// Mitsubishi GX Developer project: 11-1105_20130914   PLC: FX3U

PROGRAM MAIN
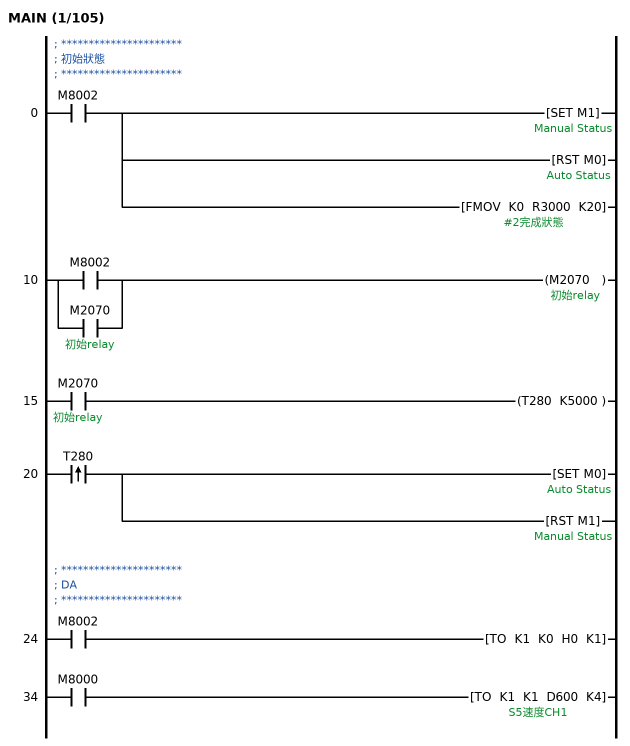
; **********************
; 初始狀態
; **********************
0     LD      M8002
      SET     M1  ; Manual Status
      RST     M0  ; Auto Status
      FMOV    K0 R3000 K20  ; #2完成狀態
10    LD      M8002
      OR      M2070  ; 初始relay
      OUT     M2070  ; 初始relay
15    LD      M2070  ; 初始relay
      OUT     T280 K5000
20    LDP     T280
      SET     M0  ; Auto Status
      RST     M1  ; Manual Status
; **********************
; DA
; **********************
24    LD      M8002
      TO      K1 K0 H0 K1
34    LD      M8000
      TO      K1 K1 D600 K4  ; S5速度CH1
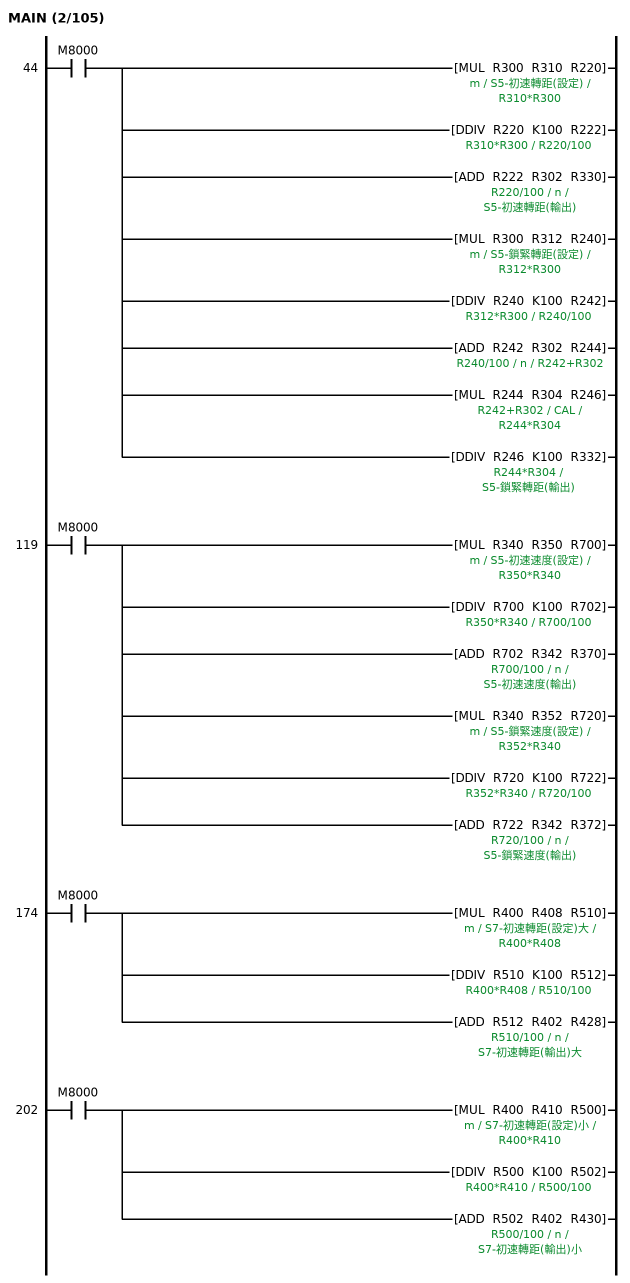
44    LD      M8000
      MUL     R300 R310 R220  ; m / S5-初速轉距(設定) / R310*R300
      DDIV    R220 K100 R222  ; R220/100
      ADD     R222 R302 R330  ; n / S5-初速轉距(輸出)
      MUL     R300 R312 R240  ; S5-鎖緊轉距(設定) / R312*R300
      DDIV    R240 K100 R242  ; R240/100
      ADD     R242 R302 R244  ; R242+R302
      MUL     R244 R304 R246  ; CAL / R244*R304
      DDIV    R246 K100 R332  ; S5-鎖緊轉距(輸出)
119   LD      M8000
      MUL     R340 R350 R700  ; m / S5-初速速度(設定) / R350*R340
      DDIV    R700 K100 R702  ; R700/100
      ADD     R702 R342 R370  ; n / S5-初速速度(輸出)
      MUL     R340 R352 R720  ; S5-鎖緊速度(設定) / R352*R340
      DDIV    R720 K100 R722  ; R720/100
      ADD     R722 R342 R372  ; S5-鎖緊速度(輸出)
174   LD      M8000
      MUL     R400 R408 R510  ; m / S7-初速轉距(設定)大 / R400*R408
      DDIV    R510 K100 R512  ; R510/100
      ADD     R512 R402 R428  ; n / S7-初速轉距(輸出)大
202   LD      M8000
      MUL     R400 R410 R500  ; S7-初速轉距(設定)小 / R400*R410
      DDIV    R500 K100 R502  ; R500/100
      ADD     R502 R402 R430  ; S7-初速轉距(輸出)小
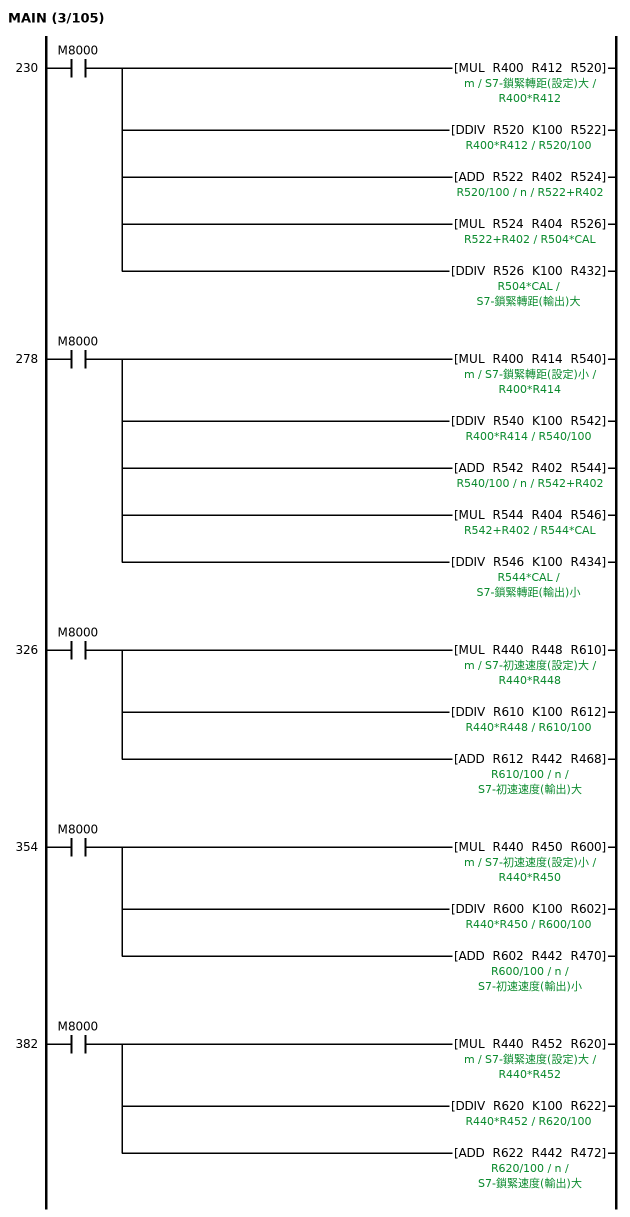
230   LD      M8000
      MUL     R400 R412 R520  ; S7-鎖緊轉距(設定)大 / R400*R412
      DDIV    R520 K100 R522  ; R520/100
      ADD     R522 R402 R524  ; R522+R402
      MUL     R524 R404 R526  ; R504*CAL
      DDIV    R526 K100 R432  ; S7-鎖緊轉距(輸出)大
278   LD      M8000
      MUL     R400 R414 R540  ; S7-鎖緊轉距(設定)小 / R400*R414
      DDIV    R540 K100 R542  ; R540/100
      ADD     R542 R402 R544  ; R542+R402
      MUL     R544 R404 R546  ; R544*CAL
      DDIV    R546 K100 R434  ; S7-鎖緊轉距(輸出)小
326   LD      M8000
      MUL     R440 R448 R610  ; m / S7-初速速度(設定)大 / R440*R448
      DDIV    R610 K100 R612  ; R610/100
      ADD     R612 R442 R468  ; n / S7-初速速度(輸出)大
354   LD      M8000
      MUL     R440 R450 R600  ; S7-初速速度(設定)小 / R440*R450
      DDIV    R600 K100 R602  ; R600/100
      ADD     R602 R442 R470  ; S7-初速速度(輸出)小
382   LD      M8000
      MUL     R440 R452 R620  ; S7-鎖緊速度(設定)大 / R440*R452
      DDIV    R620 K100 R622  ; R620/100
      ADD     R622 R442 R472  ; S7-鎖緊速度(輸出)大
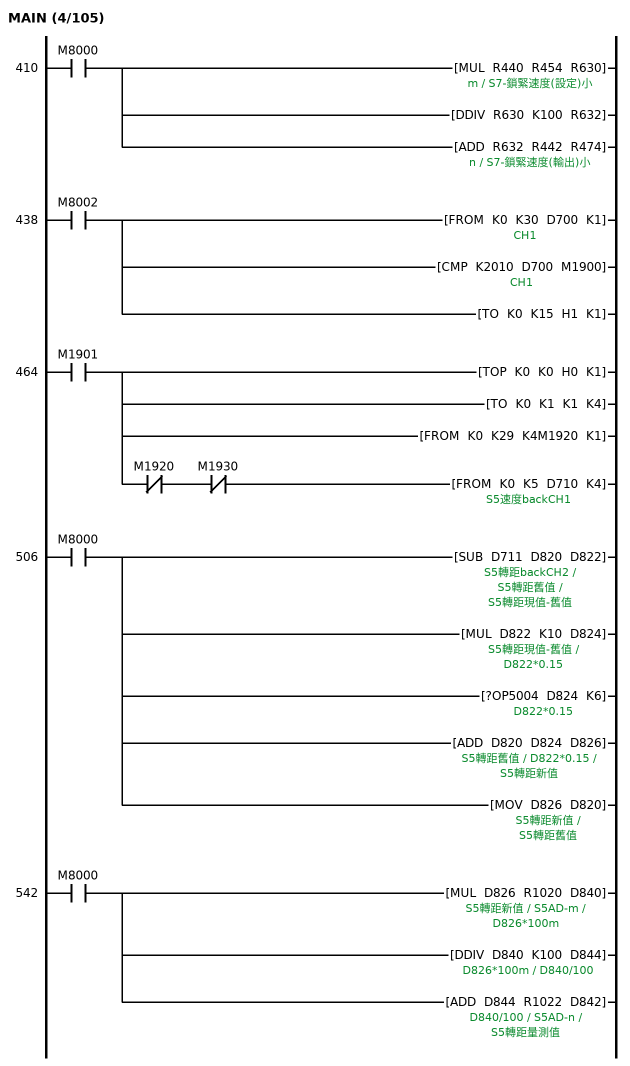
410   LD      M8000
      MUL     R440 R454 R630  ; S7-鎖緊速度(設定)小
      DDIV    R630 K100 R632
      ADD     R632 R442 R474  ; S7-鎖緊速度(輸出)小
438   LD      M8002
      FROM    K0 K30 D700 K1  ; CH1
      CMP     K2010 D700 M1900
      TO      K0 K15 H1 K1
464   LD      M1901
      TOP     K0 K0 H0 K1
      TO      K0 K1 K1 K4
      FROM    K0 K29 K4M1920 K1
      ANI     M1920
      ANI     M1930
      FROM    K0 K5 D710 K4  ; S5速度backCH1
506   LD      M8000
      SUB     D711 D820 D822  ; S5轉距backCH2 / S5轉距舊值 / S5轉距現值-舊值
      MUL     D822 K10 D824  ; D822*0.15
      ?OP5004 D824 K6
      ADD     D820 D824 D826  ; S5轉距新值
      MOV     D826 D820
542   LD      M8000
      MUL     D826 R1020 D840  ; S5AD-m / D826*100m
      DDIV    D840 K100 D844  ; D840/100
      ADD     D844 R1022 D842  ; S5AD-n / S5轉距量測值
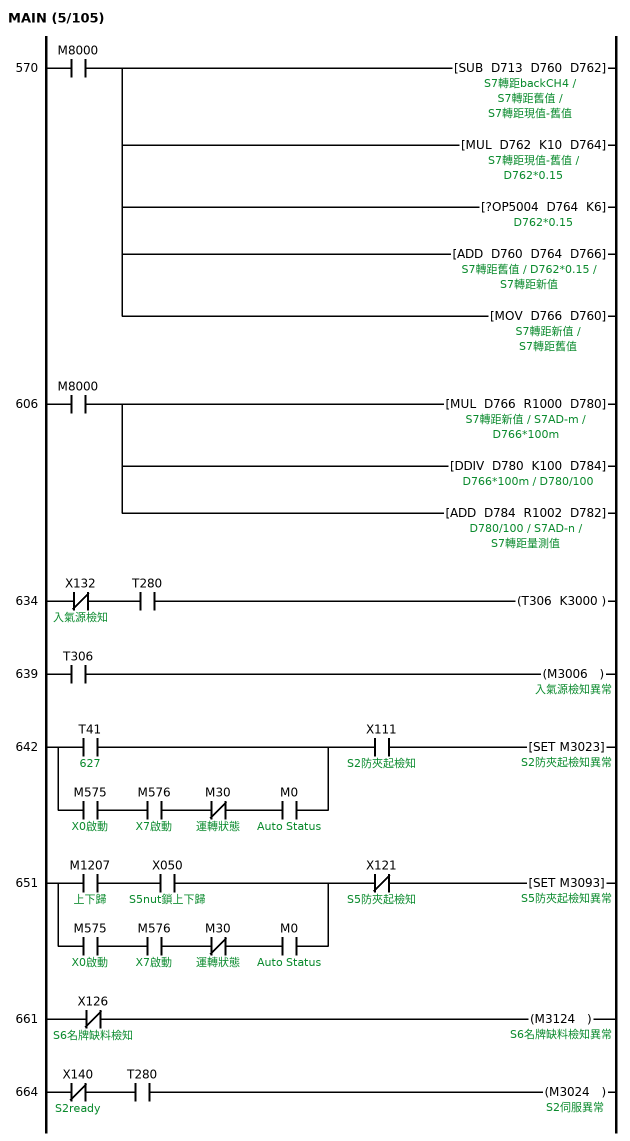
570   LD      M8000
      SUB     D713 D760 D762  ; S7轉距backCH4 / S7轉距舊值 / S7轉距現值-舊值
      MUL     D762 K10 D764  ; D762*0.15
      ?OP5004 D764 K6
      ADD     D760 D764 D766  ; S7轉距新值
      MOV     D766 D760
606   LD      M8000
      MUL     D766 R1000 D780  ; S7AD-m / D766*100m
      DDIV    D780 K100 D784  ; D780/100
      ADD     D784 R1002 D782  ; S7AD-n / S7轉距量測值
634   LDI     X132  ; 入氣源檢知
      AND     T280
      OUT     T306 K3000
639   LD      T306
      OUT     M3006  ; 入氣源檢知異常
642   LD      T41  ; 627
      LD      M575  ; X0啟動
      AND     M576  ; X7啟動
      ANI     M30  ; 運轉狀態
      AND     M0  ; Auto Status
      ORB
      AND     X111  ; S2防夾起檢知
      SET     M3023  ; S2防夾起檢知異常
651   LD      M1207  ; 上下歸
      AND     X050  ; S5nut鎖上下歸
      LD      M575  ; X0啟動
      AND     M576  ; X7啟動
      ANI     M30  ; 運轉狀態
      AND     M0  ; Auto Status
      ORB
      ANI     X121  ; S5防夾起檢知
      SET     M3093  ; S5防夾起檢知異常
661   LDI     X126  ; S6名牌缺料檢知
      OUT     M3124  ; S6名牌缺料檢知異常
664   LDI     X140  ; S2ready
      AND     T280
      OUT     M3024  ; S2伺服異常
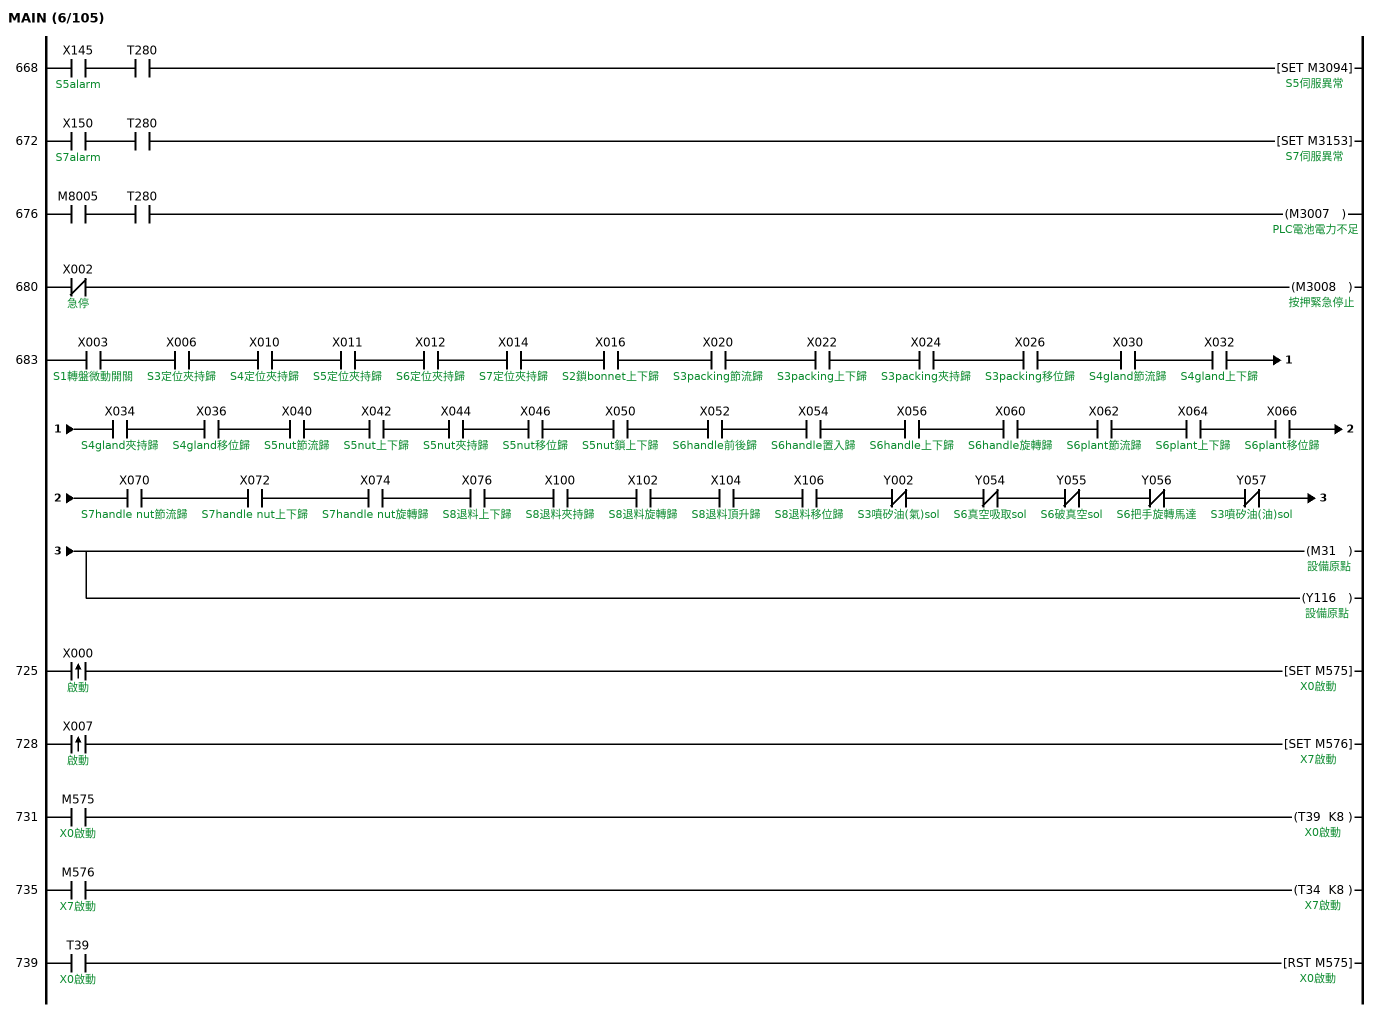
668   LD      X145  ; S5alarm
      AND     T280
      SET     M3094  ; S5伺服異常
672   LD      X150  ; S7alarm
      AND     T280
      SET     M3153  ; S7伺服異常
676   LD      M8005
      AND     T280
      OUT     M3007  ; PLC電池電力不足
680   LDI     X002  ; 急停
      OUT     M3008  ; 按押緊急停止
683   LD      X003  ; S1轉盤微動開關
      AND     X006  ; S3定位夾持歸
      AND     X010  ; S4定位夾持歸
      AND     X011  ; S5定位夾持歸
      AND     X012  ; S6定位夾持歸
      AND     X014  ; S7定位夾持歸
      AND     X016  ; S2鎖bonnet上下歸
      AND     X020  ; S3packing節流歸
      AND     X022  ; S3packing上下歸
      AND     X024  ; S3packing夾持歸
      AND     X026  ; S3packing移位歸
      AND     X030  ; S4gland節流歸
      AND     X032  ; S4gland上下歸
      AND     X034  ; S4gland夾持歸
      AND     X036  ; S4gland移位歸
      AND     X040  ; S5nut節流歸
      AND     X042  ; S5nut上下歸
      AND     X044  ; S5nut夾持歸
      AND     X046  ; S5nut移位歸
      AND     X050  ; S5nut鎖上下歸
      AND     X052  ; S6handle前後歸
      AND     X054  ; S6handle置入歸
      AND     X056  ; S6handle上下歸
      AND     X060  ; S6handle旋轉歸
      AND     X062  ; S6plant節流歸
      AND     X064  ; S6plant上下歸
      AND     X066  ; S6plant移位歸
      AND     X070  ; S7handle nut節流歸
      AND     X072  ; S7handle nut上下歸
      AND     X074  ; S7handle nut旋轉歸
      AND     X076  ; S8退料上下歸
      AND     X100  ; S8退料夾持歸
      AND     X102  ; S8退料旋轉歸
      AND     X104  ; S8退料頂升歸
      AND     X106  ; S8退料移位歸
      ANI     Y002  ; S3噴矽油(氣)sol
      ANI     Y054  ; S6真空吸取sol
      ANI     Y055  ; S6破真空sol
      ANI     Y056  ; S6把手旋轉馬達
      ANI     Y057  ; S3噴矽油(油)sol
      OUT     M31  ; 設備原點
      OUT     Y116  ; 設備原點
725   LDP     X000  ; 啟動
      SET     M575  ; X0啟動
728   LDP     X007  ; 啟動
      SET     M576  ; X7啟動
731   LD      M575  ; X0啟動
      OUT     T39 K8  ; X0啟動
735   LD      M576  ; X7啟動
      OUT     T34 K8  ; X7啟動
739   LD      T39  ; X0啟動
      RST     M575  ; X0啟動
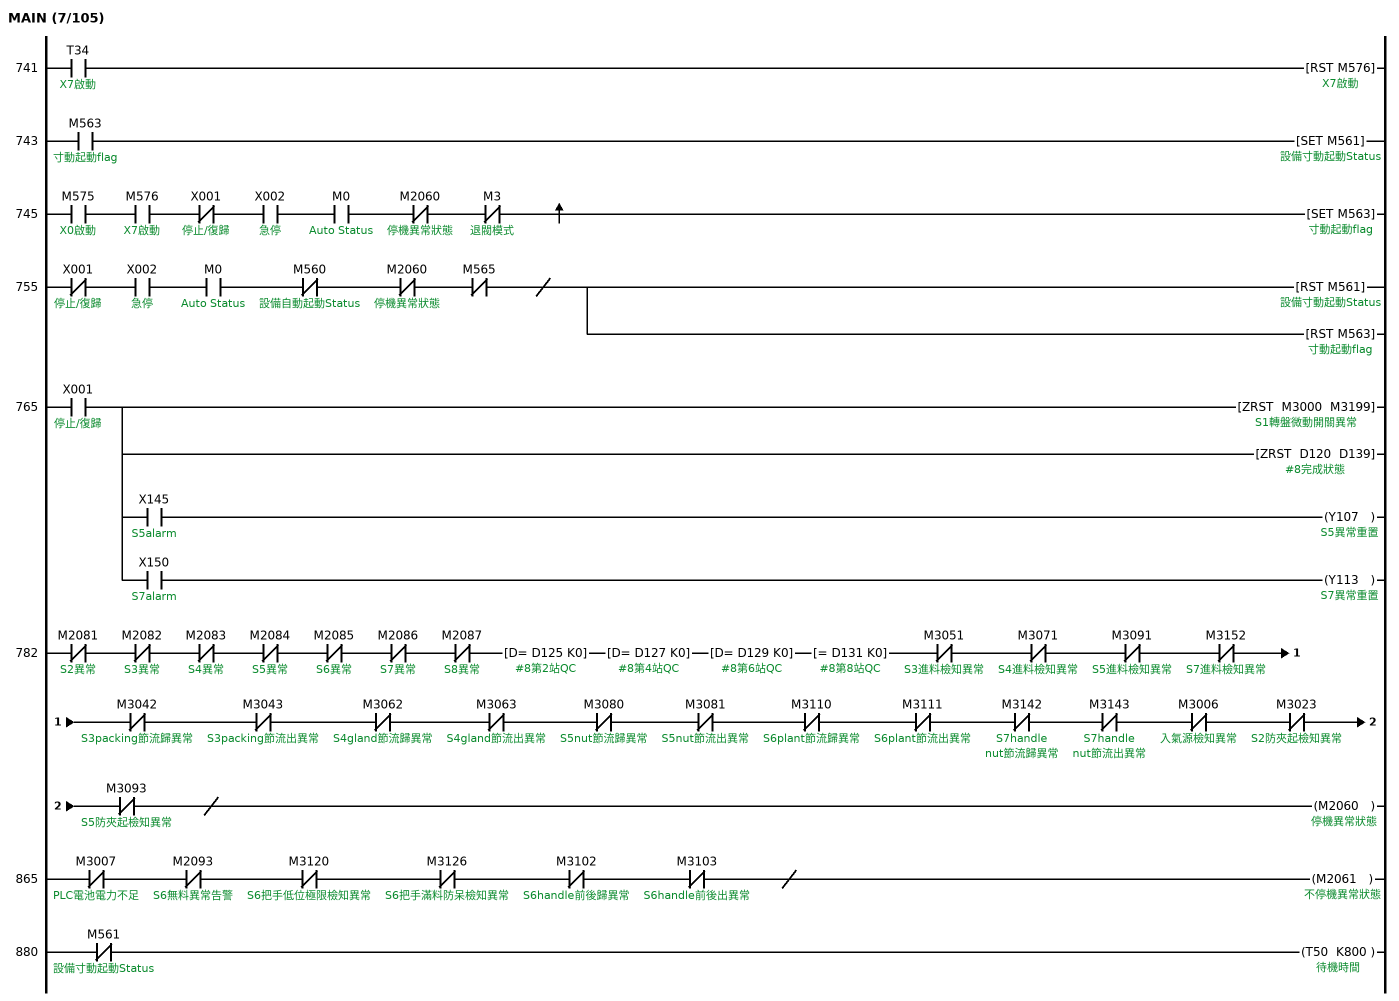
741   LD      T34  ; X7啟動
      RST     M576  ; X7啟動
743   LD      M563  ; 寸動起動flag
      SET     M561  ; 設備寸動起動Status
745   LD      M575  ; X0啟動
      AND     M576  ; X7啟動
      ANI     X001  ; 停止/復歸
      AND     X002  ; 急停
      AND     M0  ; Auto Status
      ANI     M2060  ; 停機異常狀態
      ANI     M3  ; 退閥模式
      MEP
      SET     M563  ; 寸動起動flag
755   LDI     X001  ; 停止/復歸
      AND     X002  ; 急停
      AND     M0  ; Auto Status
      ANI     M560  ; 設備自動起動Status
      ANI     M2060  ; 停機異常狀態
      ANI     M565
      INV
      RST     M561  ; 設備寸動起動Status
      RST     M563  ; 寸動起動flag
765   LD      X001  ; 停止/復歸
      ZRST    M3000 M3199  ; S1轉盤微動開關異常
      ZRST    D120 D139  ; #8完成狀態
      MPS
      AND     X145  ; S5alarm
      OUT     Y107  ; S5異常重置
      MPP
      AND     X150  ; S7alarm
      OUT     Y113  ; S7異常重置
782   LDI     M2081  ; S2異常
      ANI     M2082  ; S3異常
      ANI     M2083  ; S4異常
      ANI     M2084  ; S5異常
      ANI     M2085  ; S6異常
      ANI     M2086  ; S7異常
      ANI     M2087  ; S8異常
      ANDD=   D125 K0  ; #8第2站QC
      ANDD=   D127 K0  ; #8第4站QC
      ANDD=   D129 K0  ; #8第6站QC
      AND=    D131 K0  ; #8第8站QC
      ANI     M3051  ; S3進料檢知異常
      ANI     M3071  ; S4進料檢知異常
      ANI     M3091  ; S5進料檢知異常
      ANI     M3152  ; S7進料檢知異常
      ANI     M3042  ; S3packing節流歸異常
      ANI     M3043  ; S3packing節流出異常
      ANI     M3062  ; S4gland節流歸異常
      ANI     M3063  ; S4gland節流出異常
      ANI     M3080  ; S5nut節流歸異常
      ANI     M3081  ; S5nut節流出異常
      ANI     M3110  ; S6plant節流歸異常
      ANI     M3111  ; S6plant節流出異常
      ANI     M3142  ; S7handle nut節流歸異常
      ANI     M3143  ; S7handle nut節流出異常
      ANI     M3006  ; 入氣源檢知異常
      ANI     M3023  ; S2防夾起檢知異常
      ANI     M3093  ; S5防夾起檢知異常
      INV
      OUT     M2060  ; 停機異常狀態
865   LDI     M3007  ; PLC電池電力不足
      ANI     M2093  ; S6無料異常告警
      ANI     M3120  ; S6把手低位極限檢知異常
      ANI     M3126  ; S6把手滿料防呆檢知異常
      ANI     M3102  ; S6handle前後歸異常
      ANI     M3103  ; S6handle前後出異常
      INV
      OUT     M2061  ; 不停機異常狀態
880   LDI     M561  ; 設備寸動起動Status
      OUT     T50 K800  ; 待機時間
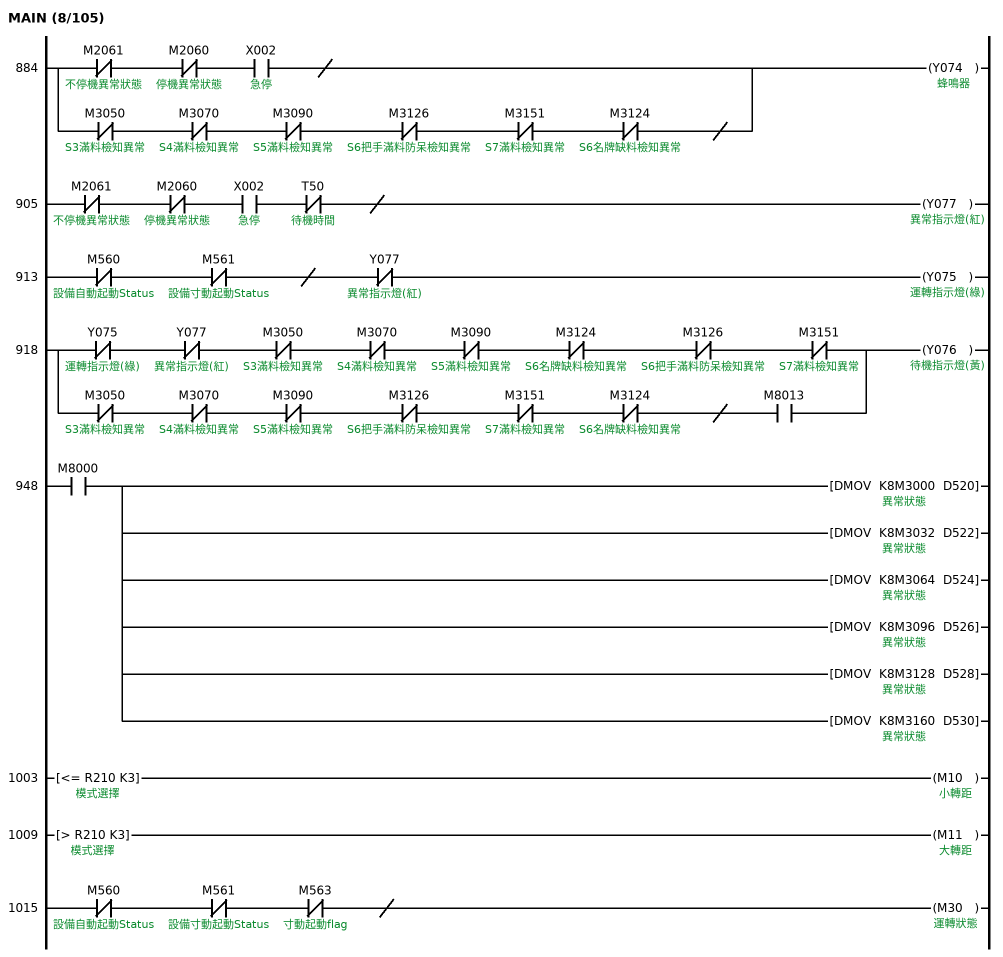
884   LDI     M2061  ; 不停機異常狀態
      ANI     M2060  ; 停機異常狀態
      AND     X002  ; 急停
      INV
      LDI     M3050  ; S3滿料檢知異常
      ANI     M3070  ; S4滿料檢知異常
      ANI     M3090  ; S5滿料檢知異常
      ANI     M3126  ; S6把手滿料防呆檢知異常
      ANI     M3151  ; S7滿料檢知異常
      ANI     M3124  ; S6名牌缺料檢知異常
      INV
      ORB
      OUT     Y074  ; 蜂鳴器
905   LDI     M2061  ; 不停機異常狀態
      ANI     M2060  ; 停機異常狀態
      AND     X002  ; 急停
      ANI     T50  ; 待機時間
      INV
      OUT     Y077  ; 異常指示燈(紅)
913   LDI     M560  ; 設備自動起動Status
      ANI     M561  ; 設備寸動起動Status
      INV
      ANI     Y077  ; 異常指示燈(紅)
      OUT     Y075  ; 運轉指示燈(綠)
918   LDI     Y075  ; 運轉指示燈(綠)
      ANI     Y077  ; 異常指示燈(紅)
      ANI     M3050  ; S3滿料檢知異常
      ANI     M3070  ; S4滿料檢知異常
      ANI     M3090  ; S5滿料檢知異常
      ANI     M3124  ; S6名牌缺料檢知異常
      ANI     M3126  ; S6把手滿料防呆檢知異常
      ANI     M3151  ; S7滿料檢知異常
      LDI     M3050  ; S3滿料檢知異常
      ANI     M3070  ; S4滿料檢知異常
      ANI     M3090  ; S5滿料檢知異常
      ANI     M3126  ; S6把手滿料防呆檢知異常
      ANI     M3151  ; S7滿料檢知異常
      ANI     M3124  ; S6名牌缺料檢知異常
      INV
      AND     M8013
      ORB
      OUT     Y076  ; 待機指示燈(黃)
948   LD      M8000
      DMOV    K8M3000 D520  ; 異常狀態
      DMOV    K8M3032 D522  ; 異常狀態
      DMOV    K8M3064 D524  ; S4gland上下歸異常 / 異常狀態
      DMOV    K8M3096 D526  ; S4定位夾持歸異常 / 異常狀態
      DMOV    K8M3128 D528  ; 異常狀態
      DMOV    K8M3160 D530  ; S8退料上下歸異常 / 異常狀態
1003  LD<=    R210 K3  ; 模式選擇
      OUT     M10  ; 小轉距
1009  LD>     R210 K3  ; 模式選擇
      OUT     M11  ; 大轉距
1015  LDI     M560  ; 設備自動起動Status
      ANI     M561  ; 設備寸動起動Status
      ANI     M563  ; 寸動起動flag
      INV
      OUT     M30  ; 運轉狀態
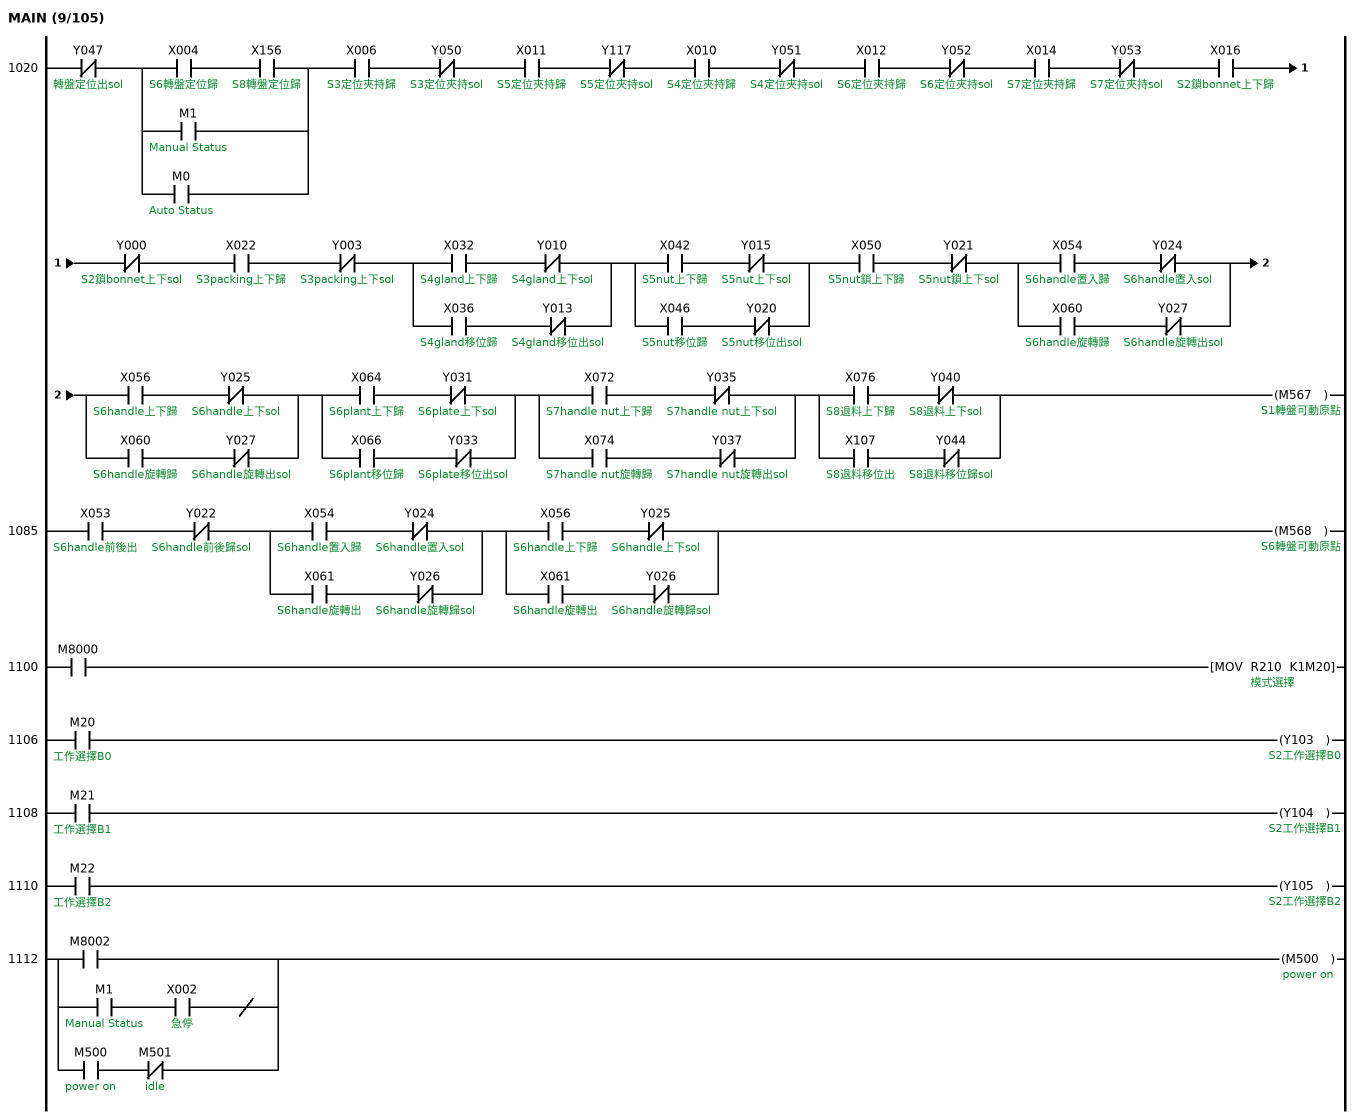
1020  LDI     Y047  ; 轉盤定位出sol
      LD      X004  ; S6轉盤定位歸
      AND     X156  ; S8轉盤定位歸
      OR      M1  ; Manual Status
      OR      M0  ; Auto Status
      ANB
      AND     X006  ; S3定位夾持歸
      ANI     Y050  ; S3定位夾持sol
      AND     X011  ; S5定位夾持歸
      ANI     Y117  ; S5定位夾持sol
      AND     X010  ; S4定位夾持歸
      ANI     Y051  ; S4定位夾持sol
      AND     X012  ; S6定位夾持歸
      ANI     Y052  ; S6定位夾持sol
      AND     X014  ; S7定位夾持歸
      ANI     Y053  ; S7定位夾持sol
      AND     X016  ; S2鎖bonnet上下歸
      ANI     Y000  ; S2鎖bonnet上下sol
      AND     X022  ; S3packing上下歸
      ANI     Y003  ; S3packing上下sol
      LD      X032  ; S4gland上下歸
      ANI     Y010  ; S4gland上下sol
      LD      X036  ; S4gland移位歸
      ANI     Y013  ; S4gland移位出sol
      ORB
      ANB
      LD      X042  ; S5nut上下歸
      ANI     Y015  ; S5nut上下sol
      LD      X046  ; S5nut移位歸
      ANI     Y020  ; S5nut移位出sol
      ORB
      ANB
      AND     X050  ; S5nut鎖上下歸
      ANI     Y021  ; S5nut鎖上下sol
      LD      X054  ; S6handle置入歸
      ANI     Y024  ; S6handle置入sol
      LD      X060  ; S6handle旋轉歸
      ANI     Y027  ; S6handle旋轉出sol
      ORB
      ANB
      LD      X056  ; S6handle上下歸
      ANI     Y025  ; S6handle上下sol
      LD      X060  ; S6handle旋轉歸
      ANI     Y027  ; S6handle旋轉出sol
      ORB
      ANB
      LD      X064  ; S6plant上下歸
      ANI     Y031  ; S6plate上下sol
      LD      X066  ; S6plant移位歸
      ANI     Y033  ; S6plate移位出sol
      ORB
      ANB
      LD      X072  ; S7handle nut上下歸
      ANI     Y035  ; S7handle nut上下sol
      LD      X074  ; S7handle nut旋轉歸
      ANI     Y037  ; S7handle nut旋轉出sol
      ORB
      ANB
      LD      X076  ; S8退料上下歸
      ANI     Y040  ; S8退料上下sol
      LD      X107  ; S8退料移位出
      ANI     Y044  ; S8退料移位歸sol
      ORB
      ANB
      OUT     M567  ; S1轉盤可動原點
1085  LD      X053  ; S6handle前後出
      ANI     Y022  ; S6handle前後歸sol
      LD      X054  ; S6handle置入歸
      ANI     Y024  ; S6handle置入sol
      LD      X061  ; S6handle旋轉出
      ANI     Y026  ; S6handle旋轉歸sol
      ORB
      ANB
      LD      X056  ; S6handle上下歸
      ANI     Y025  ; S6handle上下sol
      LD      X061  ; S6handle旋轉出
      ANI     Y026  ; S6handle旋轉歸sol
      ORB
      ANB
      OUT     M568  ; S6轉盤可動原點
1100  LD      M8000
      MOV     R210 K1M20  ; 工作選擇B0
1106  LD      M20  ; 工作選擇B0
      OUT     Y103  ; S2工作選擇B0
1108  LD      M21  ; 工作選擇B1
      OUT     Y104  ; S2工作選擇B1
1110  LD      M22  ; 工作選擇B2
      OUT     Y105  ; S2工作選擇B2
1112  LD      M8002
      LD      M1  ; Manual Status
      AND     X002  ; 急停
      INV
      ORB
      LD      M500  ; power on
      ANI     M501  ; idle
      ORB
      OUT     M500  ; power on
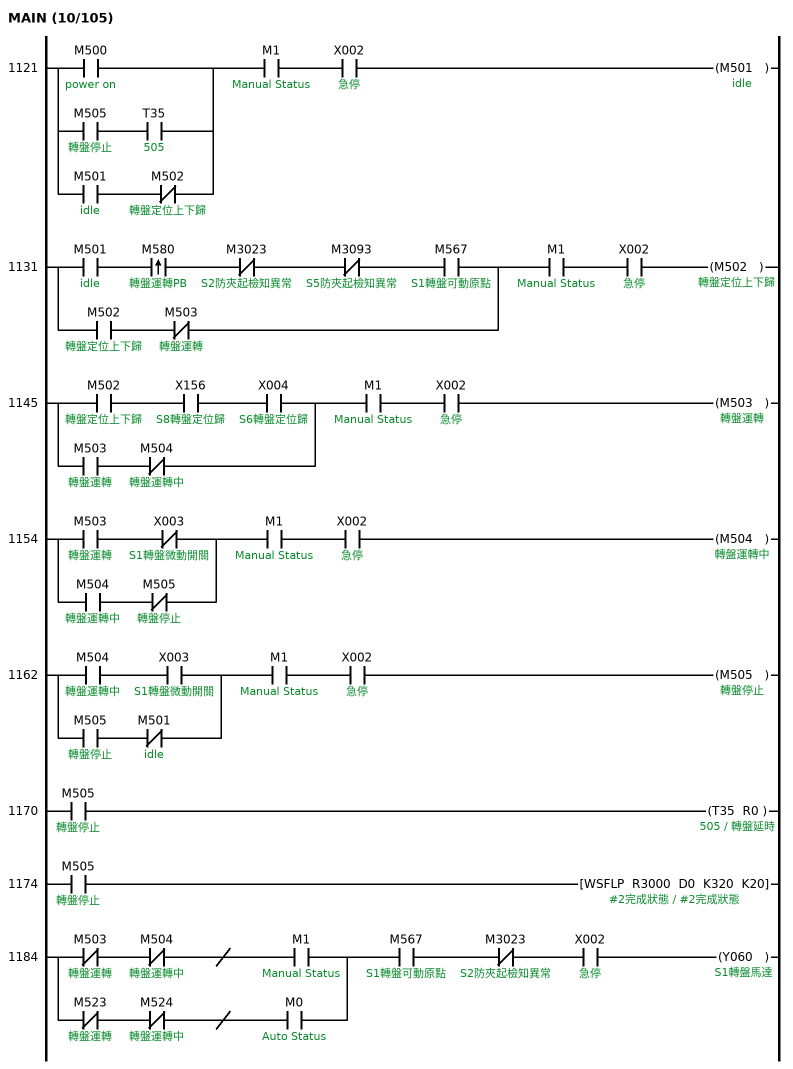
1121  LD      M500  ; power on
      LD      M505  ; 轉盤停止
      AND     T35  ; 505
      ORB
      LD      M501  ; idle
      ANI     M502  ; 轉盤定位上下歸
      ORB
      AND     M1  ; Manual Status
      AND     X002  ; 急停
      OUT     M501  ; idle
1131  LD      M501  ; idle
      ANDP    M580  ; 轉盤運轉PB
      ANI     M3023  ; S2防夾起檢知異常
      ANI     M3093  ; S5防夾起檢知異常
      AND     M567  ; S1轉盤可動原點
      LD      M502  ; 轉盤定位上下歸
      ANI     M503  ; 轉盤運轉
      ORB
      AND     M1  ; Manual Status
      AND     X002  ; 急停
      OUT     M502  ; 轉盤定位上下歸
1145  LD      M502  ; 轉盤定位上下歸
      AND     X156  ; S8轉盤定位歸
      AND     X004  ; S6轉盤定位歸
      LD      M503  ; 轉盤運轉
      ANI     M504  ; 轉盤運轉中
      ORB
      AND     M1  ; Manual Status
      AND     X002  ; 急停
      OUT     M503  ; 轉盤運轉
1154  LD      M503  ; 轉盤運轉
      ANI     X003  ; S1轉盤微動開關
      LD      M504  ; 轉盤運轉中
      ANI     M505  ; 轉盤停止
      ORB
      AND     M1  ; Manual Status
      AND     X002  ; 急停
      OUT     M504  ; 轉盤運轉中
1162  LD      M504  ; 轉盤運轉中
      AND     X003  ; S1轉盤微動開關
      LD      M505  ; 轉盤停止
      ANI     M501  ; idle
      ORB
      AND     M1  ; Manual Status
      AND     X002  ; 急停
      OUT     M505  ; 轉盤停止
1170  LD      M505  ; 轉盤停止
      OUT     T35 R0  ; 505 / 轉盤延時
1174  LD      M505  ; 轉盤停止
      WSFLP   R3000 D0 K320 K20  ; #2完成狀態
1184  LDI     M503  ; 轉盤運轉
      ANI     M504  ; 轉盤運轉中
      INV
      AND     M1  ; Manual Status
      LDI     M523  ; 轉盤運轉
      ANI     M524  ; 轉盤運轉中
      INV
      AND     M0  ; Auto Status
      ORB
      AND     M567  ; S1轉盤可動原點
      ANI     M3023  ; S2防夾起檢知異常
      AND     X002  ; 急停
      OUT     Y060  ; S1轉盤馬達
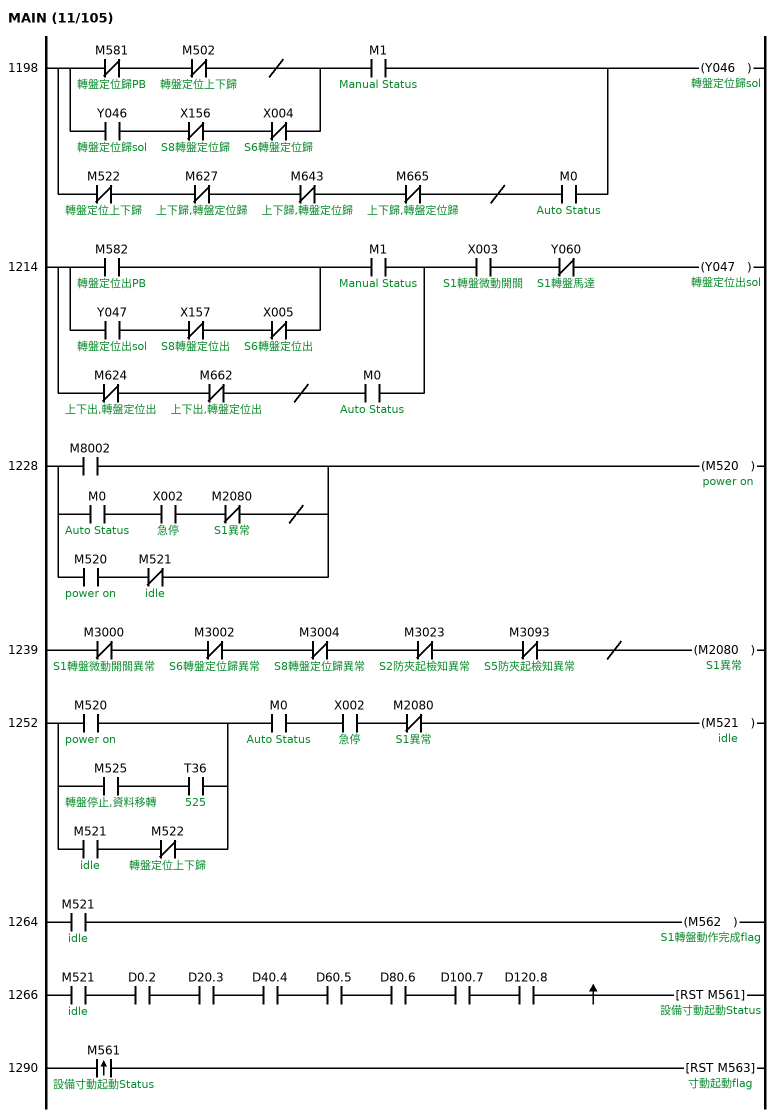
1198  LDI     M581  ; 轉盤定位歸PB
      ANI     M502  ; 轉盤定位上下歸
      INV
      LD      Y046  ; 轉盤定位歸sol
      ANI     X156  ; S8轉盤定位歸
      ANI     X004  ; S6轉盤定位歸
      ORB
      AND     M1  ; Manual Status
      LDI     M522  ; 轉盤定位上下歸
      ANI     M627  ; 上下歸,轉盤定位歸
      ANI     M643  ; 上下歸,轉盤定位歸
      ANI     M665  ; 上下歸,轉盤定位歸
      INV
      AND     M0  ; Auto Status
      ORB
      OUT     Y046  ; 轉盤定位歸sol
1214  LD      M582  ; 轉盤定位出PB
      LD      Y047  ; 轉盤定位出sol
      ANI     X157  ; S8轉盤定位出
      ANI     X005  ; S6轉盤定位出
      ORB
      AND     M1  ; Manual Status
      LDI     M624  ; 上下出,轉盤定位出
      ANI     M662  ; 上下出,轉盤定位出
      INV
      AND     M0  ; Auto Status
      ORB
      AND     X003  ; S1轉盤微動開關
      ANI     Y060  ; S1轉盤馬達
      OUT     Y047  ; 轉盤定位出sol
1228  LD      M8002
      LD      M0  ; Auto Status
      AND     X002  ; 急停
      ANI     M2080  ; S1異常
      INV
      ORB
      LD      M520  ; power on
      ANI     M521  ; idle
      ORB
      OUT     M520  ; power on
1239  LDI     M3000  ; S1轉盤微動開關異常
      ANI     M3002  ; S6轉盤定位歸異常
      ANI     M3004  ; S8轉盤定位歸異常
      ANI     M3023  ; S2防夾起檢知異常
      ANI     M3093  ; S5防夾起檢知異常
      INV
      OUT     M2080  ; S1異常
1252  LD      M520  ; power on
      LD      M525  ; 轉盤停止,資料移轉
      AND     T36  ; 525
      ORB
      LD      M521  ; idle
      ANI     M522  ; 轉盤定位上下歸
      ORB
      AND     M0  ; Auto Status
      AND     X002  ; 急停
      ANI     M2080  ; S1異常
      OUT     M521  ; idle
1264  LD      M521  ; idle
      OUT     M562  ; S1轉盤動作完成flag
1266  LD      M521  ; idle
      AND     D0.2
      AND     D20.3
      AND     D40.4
      AND     D60.5
      AND     D80.6
      AND     D100.7
      AND     D120.8
      MEP
      RST     M561  ; 設備寸動起動Status
1290  LDP     M561  ; 設備寸動起動Status
      RST     M563  ; 寸動起動flag
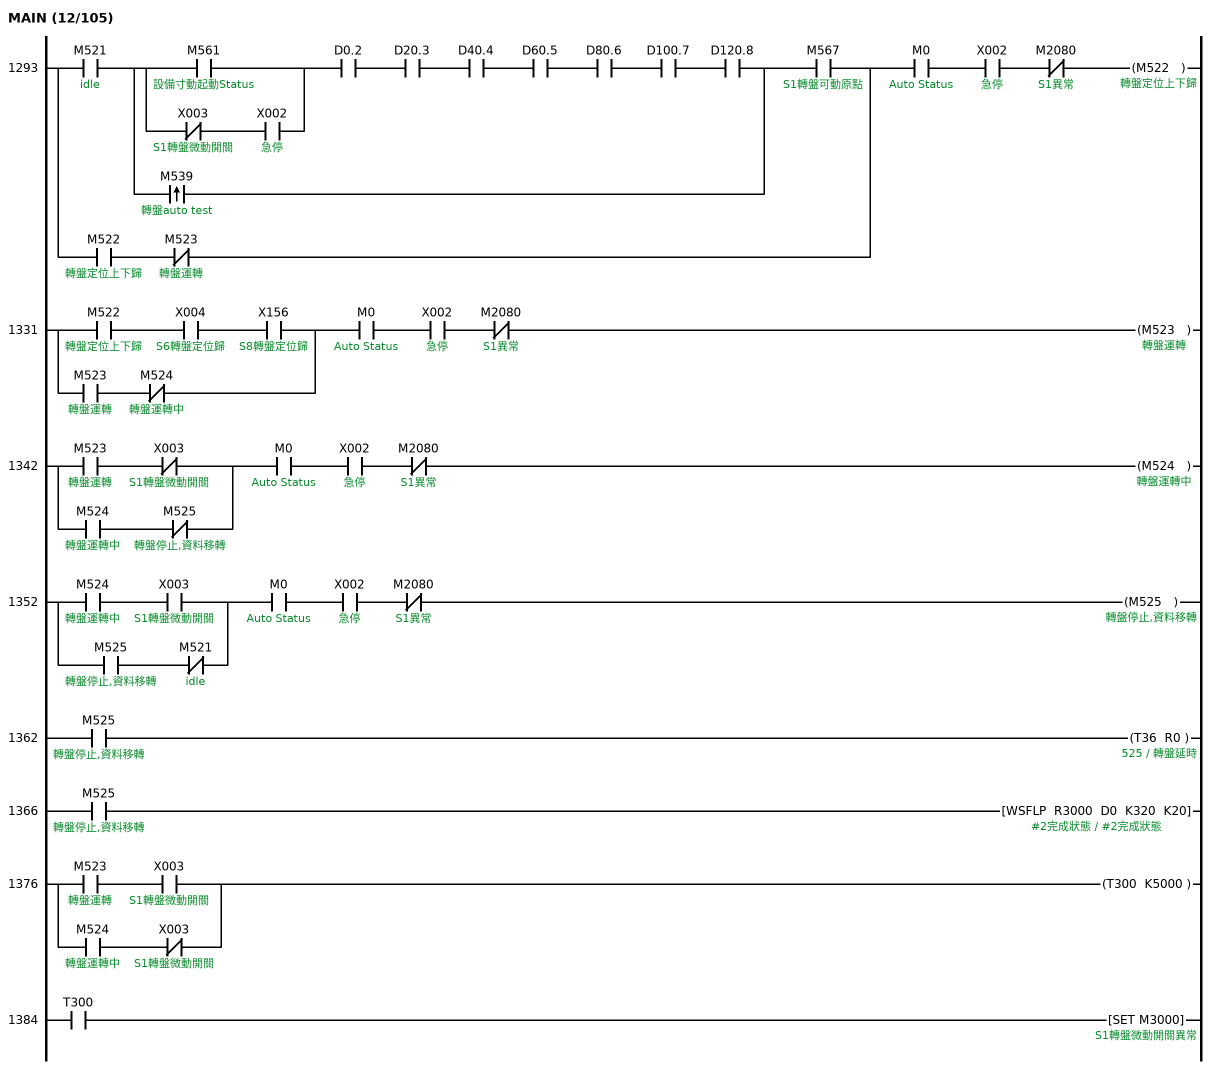
1293  LD      M521  ; idle
      LD      M561  ; 設備寸動起動Status
      LDI     X003  ; S1轉盤微動開關
      AND     X002  ; 急停
      ORB
      AND     D0.2
      AND     D20.3
      AND     D40.4
      AND     D60.5
      AND     D80.6
      AND     D100.7
      AND     D120.8
      ORP     M539  ; 轉盤auto test
      ANB
      AND     M567  ; S1轉盤可動原點
      LD      M522  ; 轉盤定位上下歸
      ANI     M523  ; 轉盤運轉
      ORB
      AND     M0  ; Auto Status
      AND     X002  ; 急停
      ANI     M2080  ; S1異常
      OUT     M522  ; 轉盤定位上下歸
1331  LD      M522  ; 轉盤定位上下歸
      AND     X004  ; S6轉盤定位歸
      AND     X156  ; S8轉盤定位歸
      LD      M523  ; 轉盤運轉
      ANI     M524  ; 轉盤運轉中
      ORB
      AND     M0  ; Auto Status
      AND     X002  ; 急停
      ANI     M2080  ; S1異常
      OUT     M523  ; 轉盤運轉
1342  LD      M523  ; 轉盤運轉
      ANI     X003  ; S1轉盤微動開關
      LD      M524  ; 轉盤運轉中
      ANI     M525  ; 轉盤停止,資料移轉
      ORB
      AND     M0  ; Auto Status
      AND     X002  ; 急停
      ANI     M2080  ; S1異常
      OUT     M524  ; 轉盤運轉中
1352  LD      M524  ; 轉盤運轉中
      AND     X003  ; S1轉盤微動開關
      LD      M525  ; 轉盤停止,資料移轉
      ANI     M521  ; idle
      ORB
      AND     M0  ; Auto Status
      AND     X002  ; 急停
      ANI     M2080  ; S1異常
      OUT     M525  ; 轉盤停止,資料移轉
1362  LD      M525  ; 轉盤停止,資料移轉
      OUT     T36 R0  ; 525 / 轉盤延時
1366  LD      M525  ; 轉盤停止,資料移轉
      WSFLP   R3000 D0 K320 K20
1376  LD      M523  ; 轉盤運轉
      AND     X003  ; S1轉盤微動開關
      LD      M524  ; 轉盤運轉中
      ANI     X003  ; S1轉盤微動開關
      ORB
      OUT     T300 K5000
1384  LD      T300
      SET     M3000  ; S1轉盤微動開關異常
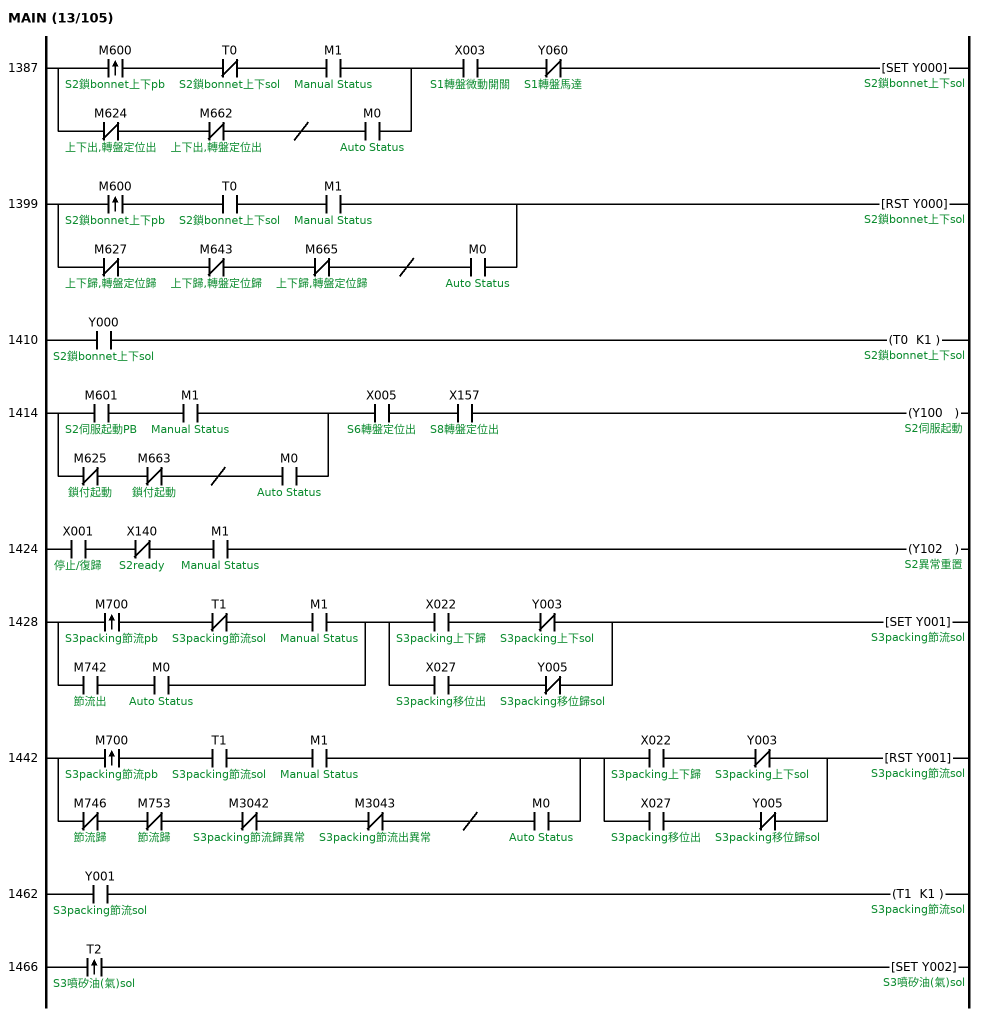
1387  LDP     M600  ; S2鎖bonnet上下pb
      ANI     T0  ; S2鎖bonnet上下sol
      AND     M1  ; Manual Status
      LDI     M624  ; 上下出,轉盤定位出
      ANI     M662  ; 上下出,轉盤定位出
      INV
      AND     M0  ; Auto Status
      ORB
      AND     X003  ; S1轉盤微動開關
      ANI     Y060  ; S1轉盤馬達
      SET     Y000  ; S2鎖bonnet上下sol
1399  LDP     M600  ; S2鎖bonnet上下pb
      AND     T0  ; S2鎖bonnet上下sol
      AND     M1  ; Manual Status
      LDI     M627  ; 上下歸,轉盤定位歸
      ANI     M643  ; 上下歸,轉盤定位歸
      ANI     M665  ; 上下歸,轉盤定位歸
      INV
      AND     M0  ; Auto Status
      ORB
      RST     Y000  ; S2鎖bonnet上下sol
1410  LD      Y000  ; S2鎖bonnet上下sol
      OUT     T0 K1  ; S2鎖bonnet上下sol
1414  LD      M601  ; S2伺服起動PB
      AND     M1  ; Manual Status
      LDI     M625  ; 鎖付起動
      ANI     M663  ; 鎖付起動
      INV
      AND     M0  ; Auto Status
      ORB
      AND     X005  ; S6轉盤定位出
      AND     X157  ; S8轉盤定位出
      OUT     Y100  ; S2伺服起動
1424  LD      X001  ; 停止/復歸
      ANI     X140  ; S2ready
      AND     M1  ; Manual Status
      OUT     Y102  ; S2異常重置
1428  LDP     M700  ; S3packing節流pb
      ANI     T1  ; S3packing節流sol
      AND     M1  ; Manual Status
      LD      M742  ; 節流出
      AND     M0  ; Auto Status
      ORB
      LD      X022  ; S3packing上下歸
      ANI     Y003  ; S3packing上下sol
      LD      X027  ; S3packing移位出
      ANI     Y005  ; S3packing移位歸sol
      ORB
      ANB
      SET     Y001  ; S3packing節流sol
1442  LDP     M700  ; S3packing節流pb
      AND     T1  ; S3packing節流sol
      AND     M1  ; Manual Status
      LDI     M746  ; 節流歸
      ANI     M753  ; 節流歸
      ANI     M3042  ; S3packing節流歸異常
      ANI     M3043  ; S3packing節流出異常
      INV
      AND     M0  ; Auto Status
      ORB
      LD      X022  ; S3packing上下歸
      ANI     Y003  ; S3packing上下sol
      LD      X027  ; S3packing移位出
      ANI     Y005  ; S3packing移位歸sol
      ORB
      ANB
      RST     Y001  ; S3packing節流sol
1462  LD      Y001  ; S3packing節流sol
      OUT     T1 K1  ; S3packing節流sol
1466  LDP     T2  ; S3噴矽油(氣)sol
      SET     Y002  ; S3噴矽油(氣)sol
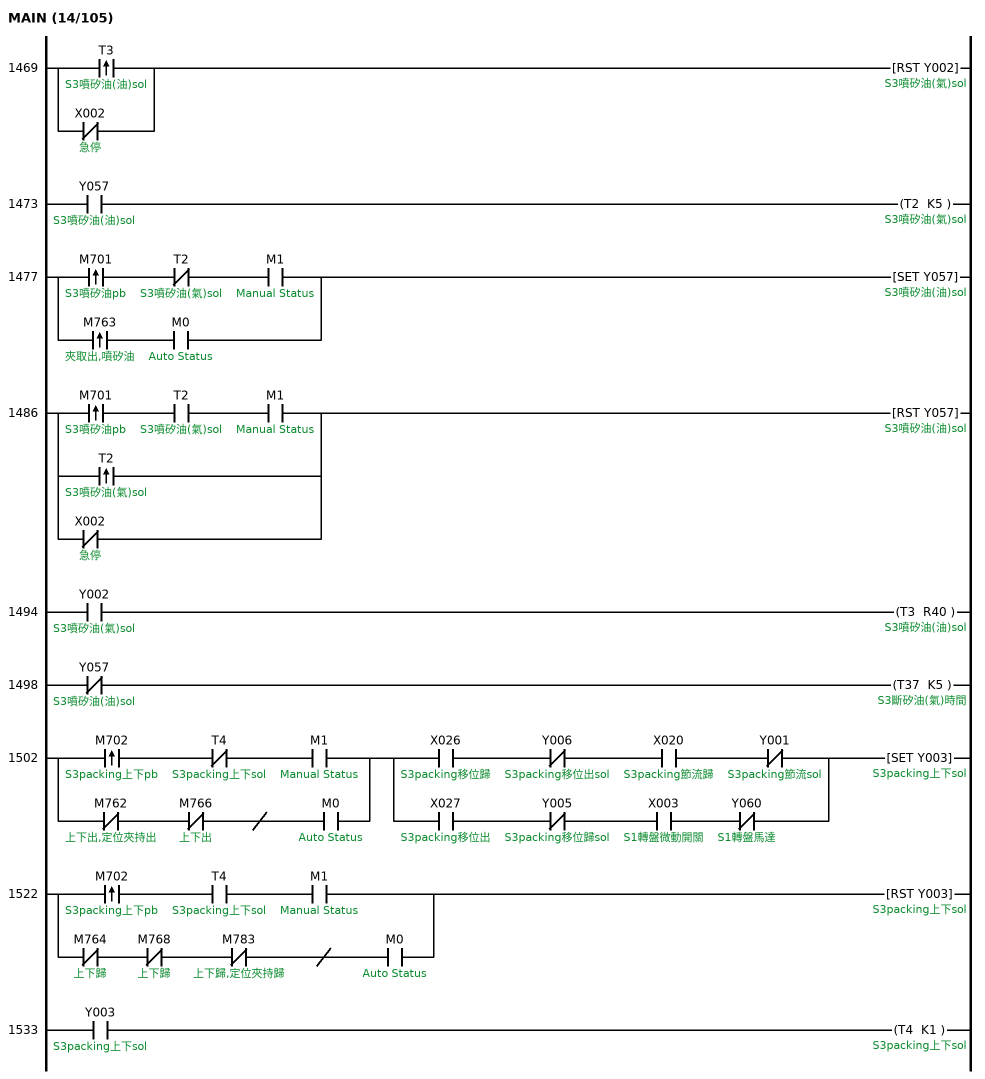
1469  LDP     T3  ; S3噴矽油(油)sol
      ORI     X002  ; 急停
      RST     Y002  ; S3噴矽油(氣)sol
1473  LD      Y057  ; S3噴矽油(油)sol
      OUT     T2 K5  ; S3噴矽油(氣)sol
1477  LDP     M701  ; S3噴矽油pb
      ANI     T2  ; S3噴矽油(氣)sol
      AND     M1  ; Manual Status
      LDP     M763  ; 夾取出,噴矽油
      AND     M0  ; Auto Status
      ORB
      SET     Y057  ; S3噴矽油(油)sol
1486  LDP     M701  ; S3噴矽油pb
      AND     T2  ; S3噴矽油(氣)sol
      AND     M1  ; Manual Status
      ORP     T2  ; S3噴矽油(氣)sol
      ORI     X002  ; 急停
      RST     Y057  ; S3噴矽油(油)sol
1494  LD      Y002  ; S3噴矽油(氣)sol
      OUT     T3 R40  ; S3噴矽油(油)sol
1498  LDI     Y057  ; S3噴矽油(油)sol
      OUT     T37 K5  ; S3斷矽油(氣)時間
1502  LDP     M702  ; S3packing上下pb
      ANI     T4  ; S3packing上下sol
      AND     M1  ; Manual Status
      LDI     M762  ; 上下出,定位夾持出
      ANI     M766  ; 上下出
      INV
      AND     M0  ; Auto Status
      ORB
      LD      X026  ; S3packing移位歸
      ANI     Y006  ; S3packing移位出sol
      AND     X020  ; S3packing節流歸
      ANI     Y001  ; S3packing節流sol
      LD      X027  ; S3packing移位出
      ANI     Y005  ; S3packing移位歸sol
      AND     X003  ; S1轉盤微動開關
      ANI     Y060  ; S1轉盤馬達
      ORB
      ANB
      SET     Y003  ; S3packing上下sol
1522  LDP     M702  ; S3packing上下pb
      AND     T4  ; S3packing上下sol
      AND     M1  ; Manual Status
      LDI     M764  ; 上下歸
      ANI     M768  ; 上下歸
      ANI     M783  ; 上下歸,定位夾持歸
      INV
      AND     M0  ; Auto Status
      ORB
      RST     Y003  ; S3packing上下sol
1533  LD      Y003  ; S3packing上下sol
      OUT     T4 K1  ; S3packing上下sol
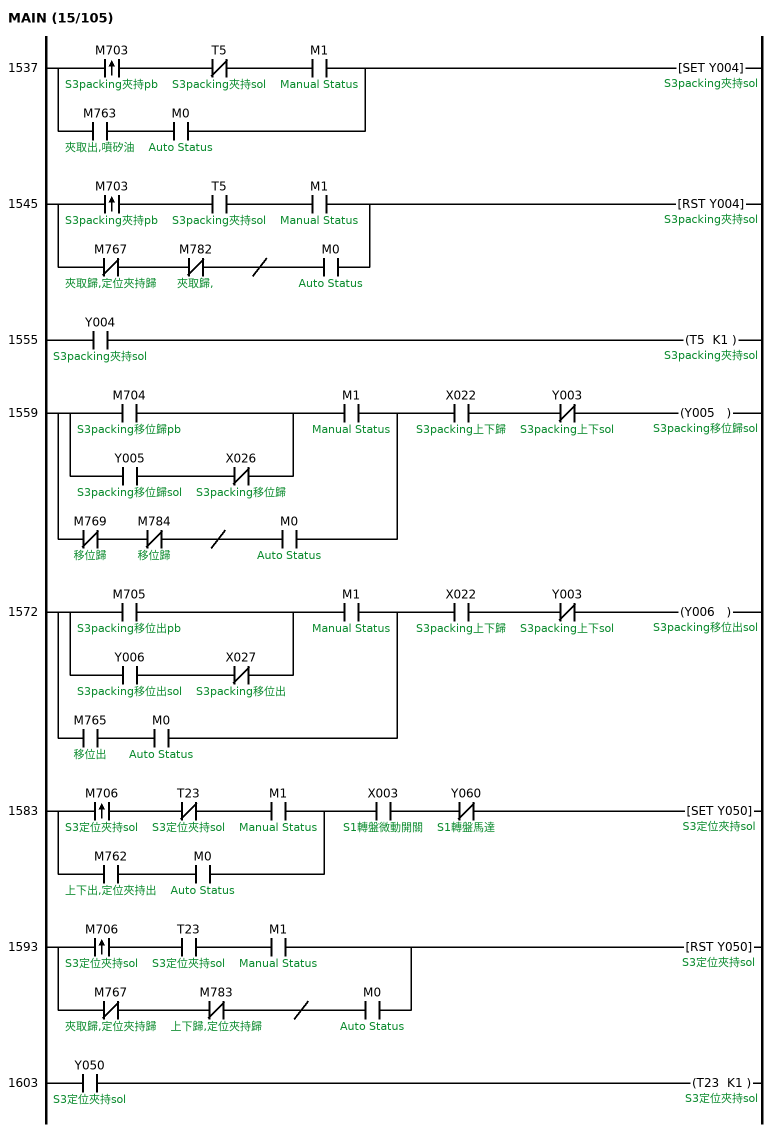
1537  LDP     M703  ; S3packing夾持pb
      ANI     T5  ; S3packing夾持sol
      AND     M1  ; Manual Status
      LD      M763  ; 夾取出,噴矽油
      AND     M0  ; Auto Status
      ORB
      SET     Y004  ; S3packing夾持sol
1545  LDP     M703  ; S3packing夾持pb
      AND     T5  ; S3packing夾持sol
      AND     M1  ; Manual Status
      LDI     M767  ; 夾取歸,定位夾持歸
      ANI     M782  ; 夾取歸,
      INV
      AND     M0  ; Auto Status
      ORB
      RST     Y004  ; S3packing夾持sol
1555  LD      Y004  ; S3packing夾持sol
      OUT     T5 K1  ; S3packing夾持sol
1559  LD      M704  ; S3packing移位歸pb
      LD      Y005  ; S3packing移位歸sol
      ANI     X026  ; S3packing移位歸
      ORB
      AND     M1  ; Manual Status
      LDI     M769  ; 移位歸
      ANI     M784  ; 移位歸
      INV
      AND     M0  ; Auto Status
      ORB
      AND     X022  ; S3packing上下歸
      ANI     Y003  ; S3packing上下sol
      OUT     Y005  ; S3packing移位歸sol
1572  LD      M705  ; S3packing移位出pb
      LD      Y006  ; S3packing移位出sol
      ANI     X027  ; S3packing移位出
      ORB
      AND     M1  ; Manual Status
      LD      M765  ; 移位出
      AND     M0  ; Auto Status
      ORB
      AND     X022  ; S3packing上下歸
      ANI     Y003  ; S3packing上下sol
      OUT     Y006  ; S3packing移位出sol
1583  LDP     M706  ; S3定位夾持sol
      ANI     T23  ; S3定位夾持sol
      AND     M1  ; Manual Status
      LD      M762  ; 上下出,定位夾持出
      AND     M0  ; Auto Status
      ORB
      AND     X003  ; S1轉盤微動開關
      ANI     Y060  ; S1轉盤馬達
      SET     Y050  ; S3定位夾持sol
1593  LDP     M706  ; S3定位夾持sol
      AND     T23  ; S3定位夾持sol
      AND     M1  ; Manual Status
      LDI     M767  ; 夾取歸,定位夾持歸
      ANI     M783  ; 上下歸,定位夾持歸
      INV
      AND     M0  ; Auto Status
      ORB
      RST     Y050  ; S3定位夾持sol
1603  LD      Y050  ; S3定位夾持sol
      OUT     T23 K1  ; S3定位夾持sol
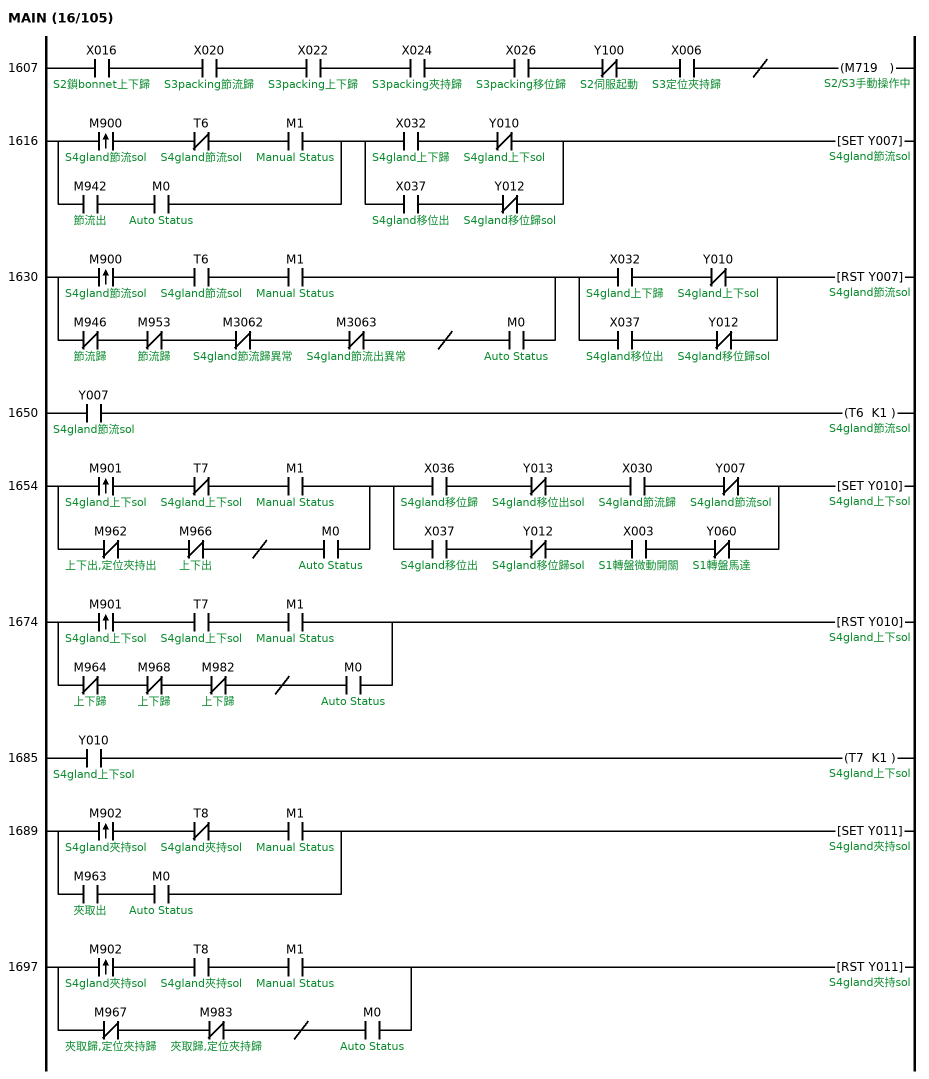
1607  LD      X016  ; S2鎖bonnet上下歸
      AND     X020  ; S3packing節流歸
      AND     X022  ; S3packing上下歸
      AND     X024  ; S3packing夾持歸
      AND     X026  ; S3packing移位歸
      ANI     Y100  ; S2伺服起動
      AND     X006  ; S3定位夾持歸
      INV
      OUT     M719  ; S2/S3手動操作中
1616  LDP     M900  ; S4gland節流sol
      ANI     T6  ; S4gland節流sol
      AND     M1  ; Manual Status
      LD      M942  ; 節流出
      AND     M0  ; Auto Status
      ORB
      LD      X032  ; S4gland上下歸
      ANI     Y010  ; S4gland上下sol
      LD      X037  ; S4gland移位出
      ANI     Y012  ; S4gland移位歸sol
      ORB
      ANB
      SET     Y007  ; S4gland節流sol
1630  LDP     M900  ; S4gland節流sol
      AND     T6  ; S4gland節流sol
      AND     M1  ; Manual Status
      LDI     M946  ; 節流歸
      ANI     M953  ; 節流歸
      ANI     M3062  ; S4gland節流歸異常
      ANI     M3063  ; S4gland節流出異常
      INV
      AND     M0  ; Auto Status
      ORB
      LD      X032  ; S4gland上下歸
      ANI     Y010  ; S4gland上下sol
      LD      X037  ; S4gland移位出
      ANI     Y012  ; S4gland移位歸sol
      ORB
      ANB
      RST     Y007  ; S4gland節流sol
1650  LD      Y007  ; S4gland節流sol
      OUT     T6 K1  ; S4gland節流sol
1654  LDP     M901  ; S4gland上下sol
      ANI     T7  ; S4gland上下sol
      AND     M1  ; Manual Status
      LDI     M962  ; 上下出,定位夾持出
      ANI     M966  ; 上下出
      INV
      AND     M0  ; Auto Status
      ORB
      LD      X036  ; S4gland移位歸
      ANI     Y013  ; S4gland移位出sol
      AND     X030  ; S4gland節流歸
      ANI     Y007  ; S4gland節流sol
      LD      X037  ; S4gland移位出
      ANI     Y012  ; S4gland移位歸sol
      AND     X003  ; S1轉盤微動開關
      ANI     Y060  ; S1轉盤馬達
      ORB
      ANB
      SET     Y010  ; S4gland上下sol
1674  LDP     M901  ; S4gland上下sol
      AND     T7  ; S4gland上下sol
      AND     M1  ; Manual Status
      LDI     M964  ; 上下歸
      ANI     M968  ; 上下歸
      ANI     M982  ; 上下歸
      INV
      AND     M0  ; Auto Status
      ORB
      RST     Y010  ; S4gland上下sol
1685  LD      Y010  ; S4gland上下sol
      OUT     T7 K1  ; S4gland上下sol
1689  LDP     M902  ; S4gland夾持sol
      ANI     T8  ; S4gland夾持sol
      AND     M1  ; Manual Status
      LD      M963  ; 夾取出
      AND     M0  ; Auto Status
      ORB
      SET     Y011  ; S4gland夾持sol
1697  LDP     M902  ; S4gland夾持sol
      AND     T8  ; S4gland夾持sol
      AND     M1  ; Manual Status
      LDI     M967  ; 夾取歸,定位夾持歸
      ANI     M983  ; 夾取歸,定位夾持歸
      INV
      AND     M0  ; Auto Status
      ORB
      RST     Y011  ; S4gland夾持sol
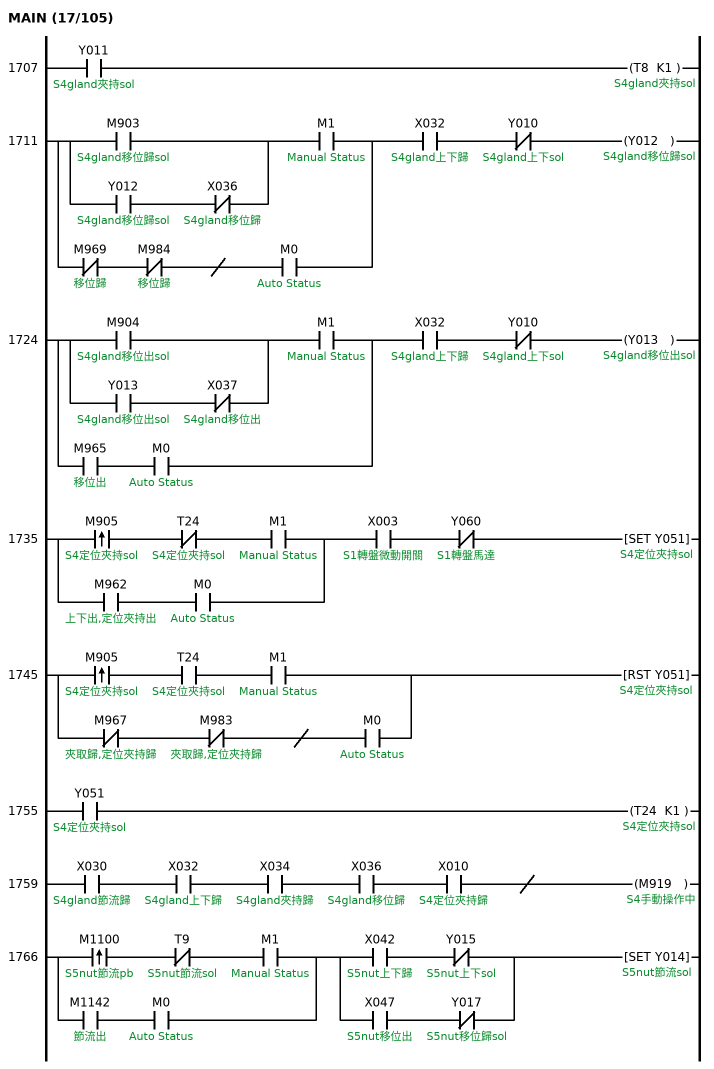
1707  LD      Y011  ; S4gland夾持sol
      OUT     T8 K1  ; S4gland夾持sol
1711  LD      M903  ; S4gland移位歸sol
      LD      Y012  ; S4gland移位歸sol
      ANI     X036  ; S4gland移位歸
      ORB
      AND     M1  ; Manual Status
      LDI     M969  ; 移位歸
      ANI     M984  ; 移位歸
      INV
      AND     M0  ; Auto Status
      ORB
      AND     X032  ; S4gland上下歸
      ANI     Y010  ; S4gland上下sol
      OUT     Y012  ; S4gland移位歸sol
1724  LD      M904  ; S4gland移位出sol
      LD      Y013  ; S4gland移位出sol
      ANI     X037  ; S4gland移位出
      ORB
      AND     M1  ; Manual Status
      LD      M965  ; 移位出
      AND     M0  ; Auto Status
      ORB
      AND     X032  ; S4gland上下歸
      ANI     Y010  ; S4gland上下sol
      OUT     Y013  ; S4gland移位出sol
1735  LDP     M905  ; S4定位夾持sol
      ANI     T24  ; S4定位夾持sol
      AND     M1  ; Manual Status
      LD      M962  ; 上下出,定位夾持出
      AND     M0  ; Auto Status
      ORB
      AND     X003  ; S1轉盤微動開關
      ANI     Y060  ; S1轉盤馬達
      SET     Y051  ; S4定位夾持sol
1745  LDP     M905  ; S4定位夾持sol
      AND     T24  ; S4定位夾持sol
      AND     M1  ; Manual Status
      LDI     M967  ; 夾取歸,定位夾持歸
      ANI     M983  ; 夾取歸,定位夾持歸
      INV
      AND     M0  ; Auto Status
      ORB
      RST     Y051  ; S4定位夾持sol
1755  LD      Y051  ; S4定位夾持sol
      OUT     T24 K1  ; S4定位夾持sol
1759  LD      X030  ; S4gland節流歸
      AND     X032  ; S4gland上下歸
      AND     X034  ; S4gland夾持歸
      AND     X036  ; S4gland移位歸
      AND     X010  ; S4定位夾持歸
      INV
      OUT     M919  ; S4手動操作中
1766  LDP     M1100  ; S5nut節流pb
      ANI     T9  ; S5nut節流sol
      AND     M1  ; Manual Status
      LD      M1142  ; 節流出
      AND     M0  ; Auto Status
      ORB
      LD      X042  ; S5nut上下歸
      ANI     Y015  ; S5nut上下sol
      LD      X047  ; S5nut移位出
      ANI     Y017  ; S5nut移位歸sol
      ORB
      ANB
      SET     Y014  ; S5nut節流sol
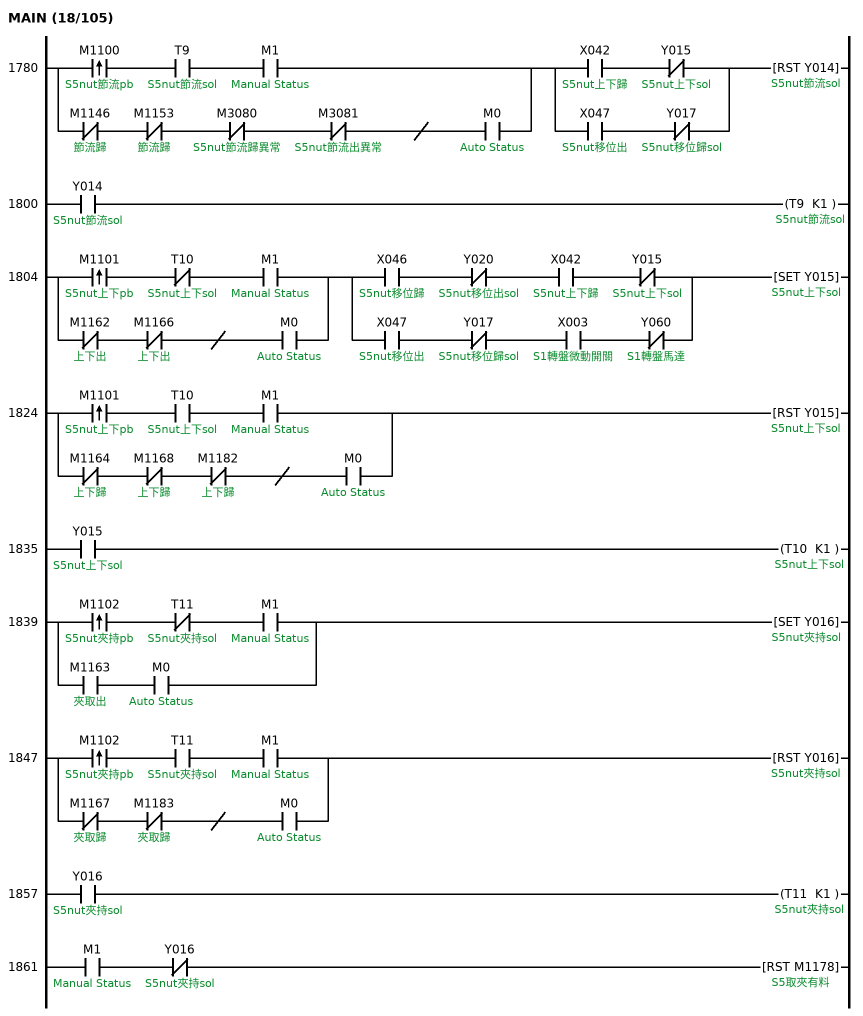
1780  LDP     M1100  ; S5nut節流pb
      AND     T9  ; S5nut節流sol
      AND     M1  ; Manual Status
      LDI     M1146  ; 節流歸
      ANI     M1153  ; 節流歸
      ANI     M3080  ; S5nut節流歸異常
      ANI     M3081  ; S5nut節流出異常
      INV
      AND     M0  ; Auto Status
      ORB
      LD      X042  ; S5nut上下歸
      ANI     Y015  ; S5nut上下sol
      LD      X047  ; S5nut移位出
      ANI     Y017  ; S5nut移位歸sol
      ORB
      ANB
      RST     Y014  ; S5nut節流sol
1800  LD      Y014  ; S5nut節流sol
      OUT     T9 K1  ; S5nut節流sol
1804  LDP     M1101  ; S5nut上下pb
      ANI     T10  ; S5nut上下sol
      AND     M1  ; Manual Status
      LDI     M1162  ; 上下出
      ANI     M1166  ; 上下出
      INV
      AND     M0  ; Auto Status
      ORB
      LD      X046  ; S5nut移位歸
      ANI     Y020  ; S5nut移位出sol
      AND     X042  ; S5nut上下歸
      ANI     Y015  ; S5nut上下sol
      LD      X047  ; S5nut移位出
      ANI     Y017  ; S5nut移位歸sol
      AND     X003  ; S1轉盤微動開關
      ANI     Y060  ; S1轉盤馬達
      ORB
      ANB
      SET     Y015  ; S5nut上下sol
1824  LDP     M1101  ; S5nut上下pb
      AND     T10  ; S5nut上下sol
      AND     M1  ; Manual Status
      LDI     M1164  ; 上下歸
      ANI     M1168  ; 上下歸
      ANI     M1182  ; 上下歸
      INV
      AND     M0  ; Auto Status
      ORB
      RST     Y015  ; S5nut上下sol
1835  LD      Y015  ; S5nut上下sol
      OUT     T10 K1  ; S5nut上下sol
1839  LDP     M1102  ; S5nut夾持pb
      ANI     T11  ; S5nut夾持sol
      AND     M1  ; Manual Status
      LD      M1163  ; 夾取出
      AND     M0  ; Auto Status
      ORB
      SET     Y016  ; S5nut夾持sol
1847  LDP     M1102  ; S5nut夾持pb
      AND     T11  ; S5nut夾持sol
      AND     M1  ; Manual Status
      LDI     M1167  ; 夾取歸
      ANI     M1183  ; 夾取歸
      INV
      AND     M0  ; Auto Status
      ORB
      RST     Y016  ; S5nut夾持sol
1857  LD      Y016  ; S5nut夾持sol
      OUT     T11 K1  ; S5nut夾持sol
1861  LD      M1  ; Manual Status
      ANI     Y016  ; S5nut夾持sol
      RST     M1178  ; S5取夾有料
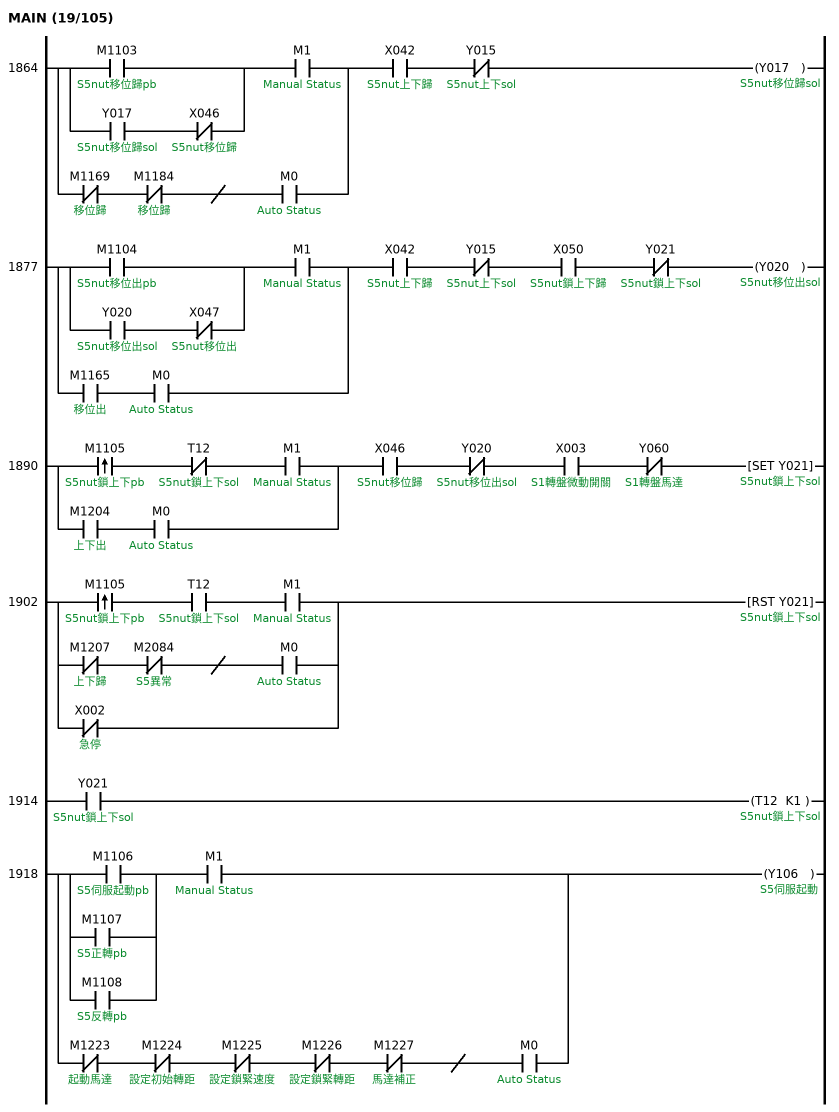
1864  LD      M1103  ; S5nut移位歸pb
      LD      Y017  ; S5nut移位歸sol
      ANI     X046  ; S5nut移位歸
      ORB
      AND     M1  ; Manual Status
      LDI     M1169  ; 移位歸
      ANI     M1184  ; 移位歸
      INV
      AND     M0  ; Auto Status
      ORB
      AND     X042  ; S5nut上下歸
      ANI     Y015  ; S5nut上下sol
      OUT     Y017  ; S5nut移位歸sol
1877  LD      M1104  ; S5nut移位出pb
      LD      Y020  ; S5nut移位出sol
      ANI     X047  ; S5nut移位出
      ORB
      AND     M1  ; Manual Status
      LD      M1165  ; 移位出
      AND     M0  ; Auto Status
      ORB
      AND     X042  ; S5nut上下歸
      ANI     Y015  ; S5nut上下sol
      AND     X050  ; S5nut鎖上下歸
      ANI     Y021  ; S5nut鎖上下sol
      OUT     Y020  ; S5nut移位出sol
1890  LDP     M1105  ; S5nut鎖上下pb
      ANI     T12  ; S5nut鎖上下sol
      AND     M1  ; Manual Status
      LD      M1204  ; 上下出
      AND     M0  ; Auto Status
      ORB
      AND     X046  ; S5nut移位歸
      ANI     Y020  ; S5nut移位出sol
      AND     X003  ; S1轉盤微動開關
      ANI     Y060  ; S1轉盤馬達
      SET     Y021  ; S5nut鎖上下sol
1902  LDP     M1105  ; S5nut鎖上下pb
      AND     T12  ; S5nut鎖上下sol
      AND     M1  ; Manual Status
      LDI     M1207  ; 上下歸
      ANI     M2084  ; S5異常
      INV
      AND     M0  ; Auto Status
      ORB
      ORI     X002  ; 急停
      RST     Y021  ; S5nut鎖上下sol
1914  LD      Y021  ; S5nut鎖上下sol
      OUT     T12 K1  ; S5nut鎖上下sol
1918  LD      M1106  ; S5伺服起動pb
      OR      M1107  ; S5正轉pb
      OR      M1108  ; S5反轉pb
      AND     M1  ; Manual Status
      LDI     M1223  ; 起動馬達
      ANI     M1224  ; 設定初始轉距
      ANI     M1225  ; 設定鎖緊速度
      ANI     M1226  ; 設定鎖緊轉距
      ANI     M1227  ; 馬達補正
      INV
      AND     M0  ; Auto Status
      ORB
      OUT     Y106  ; S5伺服起動
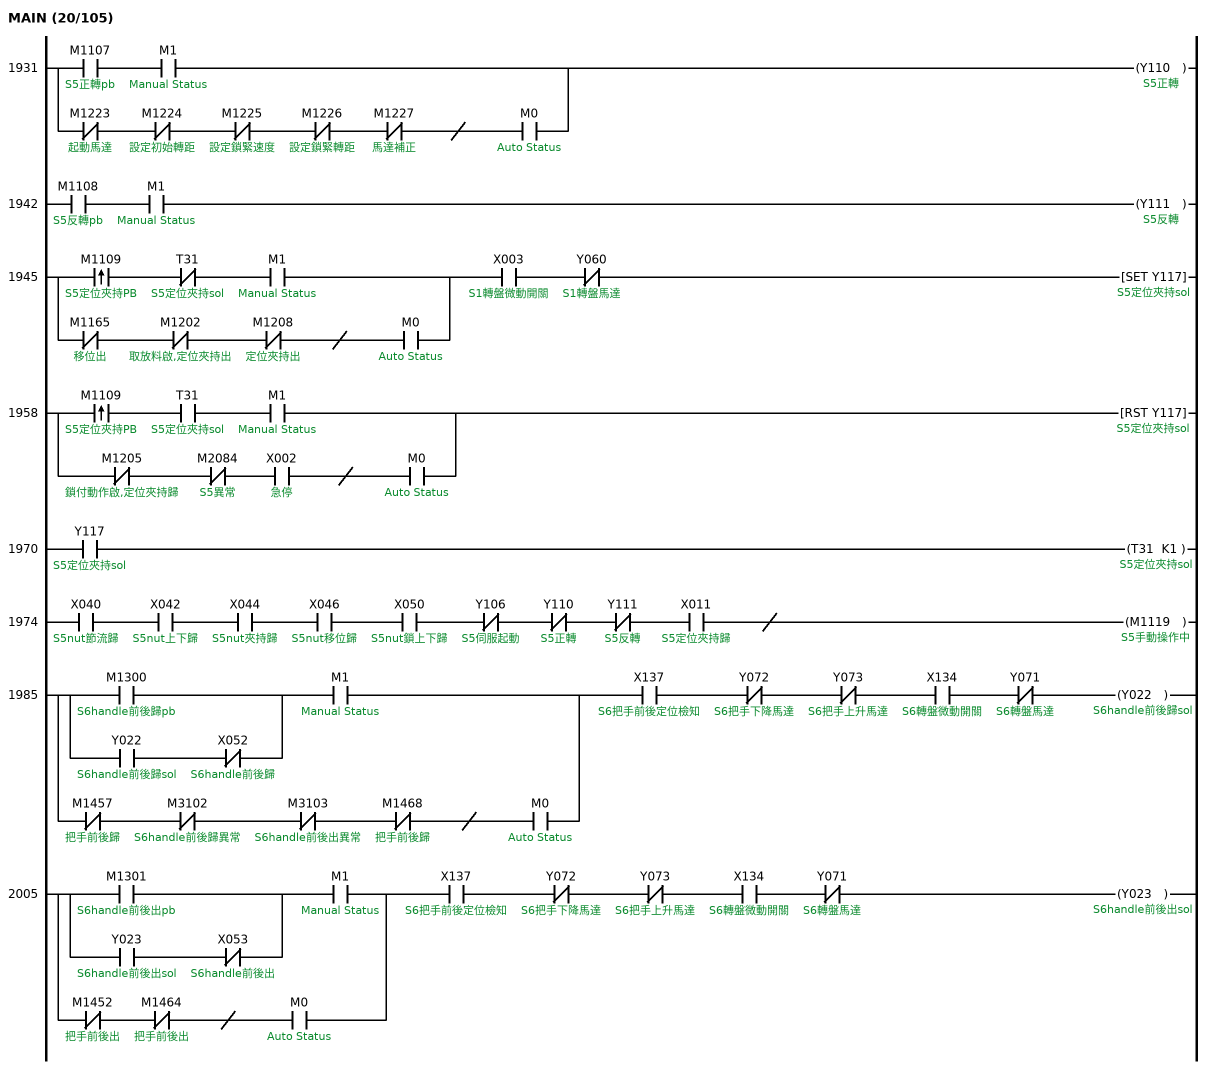
1931  LD      M1107  ; S5正轉pb
      AND     M1  ; Manual Status
      LDI     M1223  ; 起動馬達
      ANI     M1224  ; 設定初始轉距
      ANI     M1225  ; 設定鎖緊速度
      ANI     M1226  ; 設定鎖緊轉距
      ANI     M1227  ; 馬達補正
      INV
      AND     M0  ; Auto Status
      ORB
      OUT     Y110  ; S5正轉
1942  LD      M1108  ; S5反轉pb
      AND     M1  ; Manual Status
      OUT     Y111  ; S5反轉
1945  LDP     M1109  ; S5定位夾持PB
      ANI     T31  ; S5定位夾持sol
      AND     M1  ; Manual Status
      LDI     M1165  ; 移位出
      ANI     M1202  ; 取放料啟,定位夾持出
      ANI     M1208  ; 定位夾持出
      INV
      AND     M0  ; Auto Status
      ORB
      AND     X003  ; S1轉盤微動開關
      ANI     Y060  ; S1轉盤馬達
      SET     Y117  ; S5定位夾持sol
1958  LDP     M1109  ; S5定位夾持PB
      AND     T31  ; S5定位夾持sol
      AND     M1  ; Manual Status
      LDI     M1205  ; 鎖付動作啟,定位夾持歸
      ANI     M2084  ; S5異常
      AND     X002  ; 急停
      INV
      AND     M0  ; Auto Status
      ORB
      RST     Y117  ; S5定位夾持sol
1970  LD      Y117  ; S5定位夾持sol
      OUT     T31 K1  ; S5定位夾持sol
1974  LD      X040  ; S5nut節流歸
      AND     X042  ; S5nut上下歸
      AND     X044  ; S5nut夾持歸
      AND     X046  ; S5nut移位歸
      AND     X050  ; S5nut鎖上下歸
      ANI     Y106  ; S5伺服起動
      ANI     Y110  ; S5正轉
      ANI     Y111  ; S5反轉
      AND     X011  ; S5定位夾持歸
      INV
      OUT     M1119  ; S5手動操作中
1985  LD      M1300  ; S6handle前後歸pb
      LD      Y022  ; S6handle前後歸sol
      ANI     X052  ; S6handle前後歸
      ORB
      AND     M1  ; Manual Status
      LDI     M1457  ; 把手前後歸
      ANI     M3102  ; S6handle前後歸異常
      ANI     M3103  ; S6handle前後出異常
      ANI     M1468  ; 把手前後歸
      INV
      AND     M0  ; Auto Status
      ORB
      AND     X137  ; S6把手前後定位檢知
      ANI     Y072  ; S6把手下降馬達
      ANI     Y073  ; S6把手上升馬達
      AND     X134  ; S6轉盤微動開關
      ANI     Y071  ; S6轉盤馬達
      OUT     Y022  ; S6handle前後歸sol
2005  LD      M1301  ; S6handle前後出pb
      LD      Y023  ; S6handle前後出sol
      ANI     X053  ; S6handle前後出
      ORB
      AND     M1  ; Manual Status
      LDI     M1452  ; 把手前後出
      ANI     M1464  ; 把手前後出
      INV
      AND     M0  ; Auto Status
      ORB
      AND     X137  ; S6把手前後定位檢知
      ANI     Y072  ; S6把手下降馬達
      ANI     Y073  ; S6把手上升馬達
      AND     X134  ; S6轉盤微動開關
      ANI     Y071  ; S6轉盤馬達
      OUT     Y023  ; S6handle前後出sol
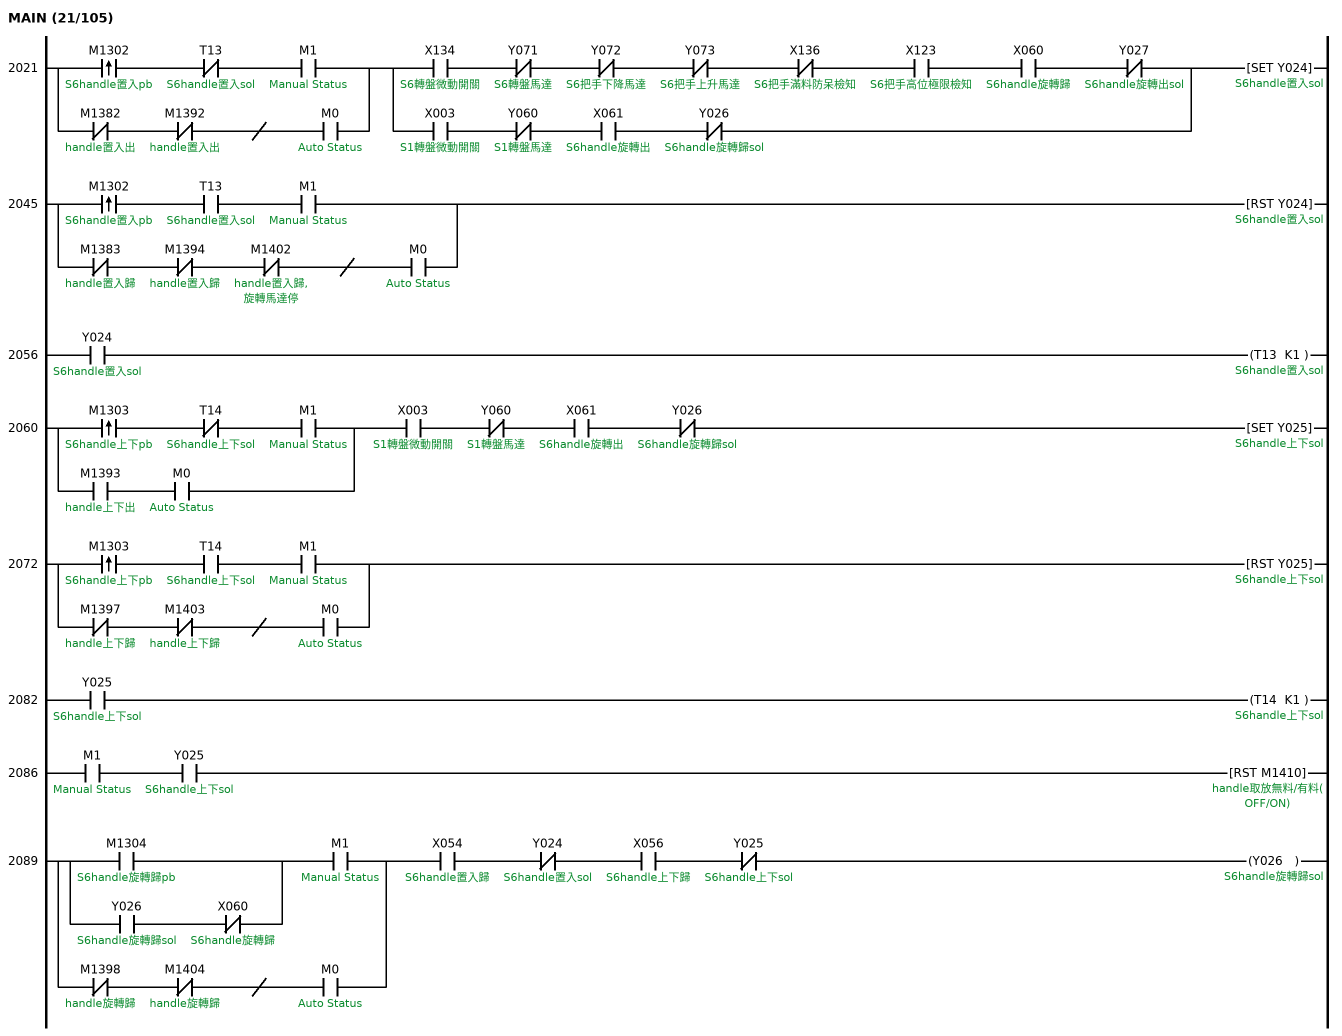
2021  LDP     M1302  ; S6handle置入pb
      ANI     T13  ; S6handle置入sol
      AND     M1  ; Manual Status
      LDI     M1382  ; handle置入出
      ANI     M1392  ; handle置入出
      INV
      AND     M0  ; Auto Status
      ORB
      LD      X134  ; S6轉盤微動開關
      ANI     Y071  ; S6轉盤馬達
      ANI     Y072  ; S6把手下降馬達
      ANI     Y073  ; S6把手上升馬達
      ANI     X136  ; S6把手滿料防呆檢知
      AND     X123  ; S6把手高位極限檢知
      AND     X060  ; S6handle旋轉歸
      ANI     Y027  ; S6handle旋轉出sol
      LD      X003  ; S1轉盤微動開關
      ANI     Y060  ; S1轉盤馬達
      AND     X061  ; S6handle旋轉出
      ANI     Y026  ; S6handle旋轉歸sol
      ORB
      ANB
      SET     Y024  ; S6handle置入sol
2045  LDP     M1302  ; S6handle置入pb
      AND     T13  ; S6handle置入sol
      AND     M1  ; Manual Status
      LDI     M1383  ; handle置入歸
      ANI     M1394  ; handle置入歸
      ANI     M1402  ; handle置入歸,旋轉馬達停
      INV
      AND     M0  ; Auto Status
      ORB
      RST     Y024  ; S6handle置入sol
2056  LD      Y024  ; S6handle置入sol
      OUT     T13 K1  ; S6handle置入sol
2060  LDP     M1303  ; S6handle上下pb
      ANI     T14  ; S6handle上下sol
      AND     M1  ; Manual Status
      LD      M1393  ; handle上下出
      AND     M0  ; Auto Status
      ORB
      AND     X003  ; S1轉盤微動開關
      ANI     Y060  ; S1轉盤馬達
      AND     X061  ; S6handle旋轉出
      ANI     Y026  ; S6handle旋轉歸sol
      SET     Y025  ; S6handle上下sol
2072  LDP     M1303  ; S6handle上下pb
      AND     T14  ; S6handle上下sol
      AND     M1  ; Manual Status
      LDI     M1397  ; handle上下歸
      ANI     M1403  ; handle上下歸
      INV
      AND     M0  ; Auto Status
      ORB
      RST     Y025  ; S6handle上下sol
2082  LD      Y025  ; S6handle上下sol
      OUT     T14 K1  ; S6handle上下sol
2086  LD      M1  ; Manual Status
      AND     Y025  ; S6handle上下sol
      RST     M1410  ; handle取放無料/有料(OFF/ON)
2089  LD      M1304  ; S6handle旋轉歸pb
      LD      Y026  ; S6handle旋轉歸sol
      ANI     X060  ; S6handle旋轉歸
      ORB
      AND     M1  ; Manual Status
      LDI     M1398  ; handle旋轉歸
      ANI     M1404  ; handle旋轉歸
      INV
      AND     M0  ; Auto Status
      ORB
      AND     X054  ; S6handle置入歸
      ANI     Y024  ; S6handle置入sol
      AND     X056  ; S6handle上下歸
      ANI     Y025  ; S6handle上下sol
      OUT     Y026  ; S6handle旋轉歸sol
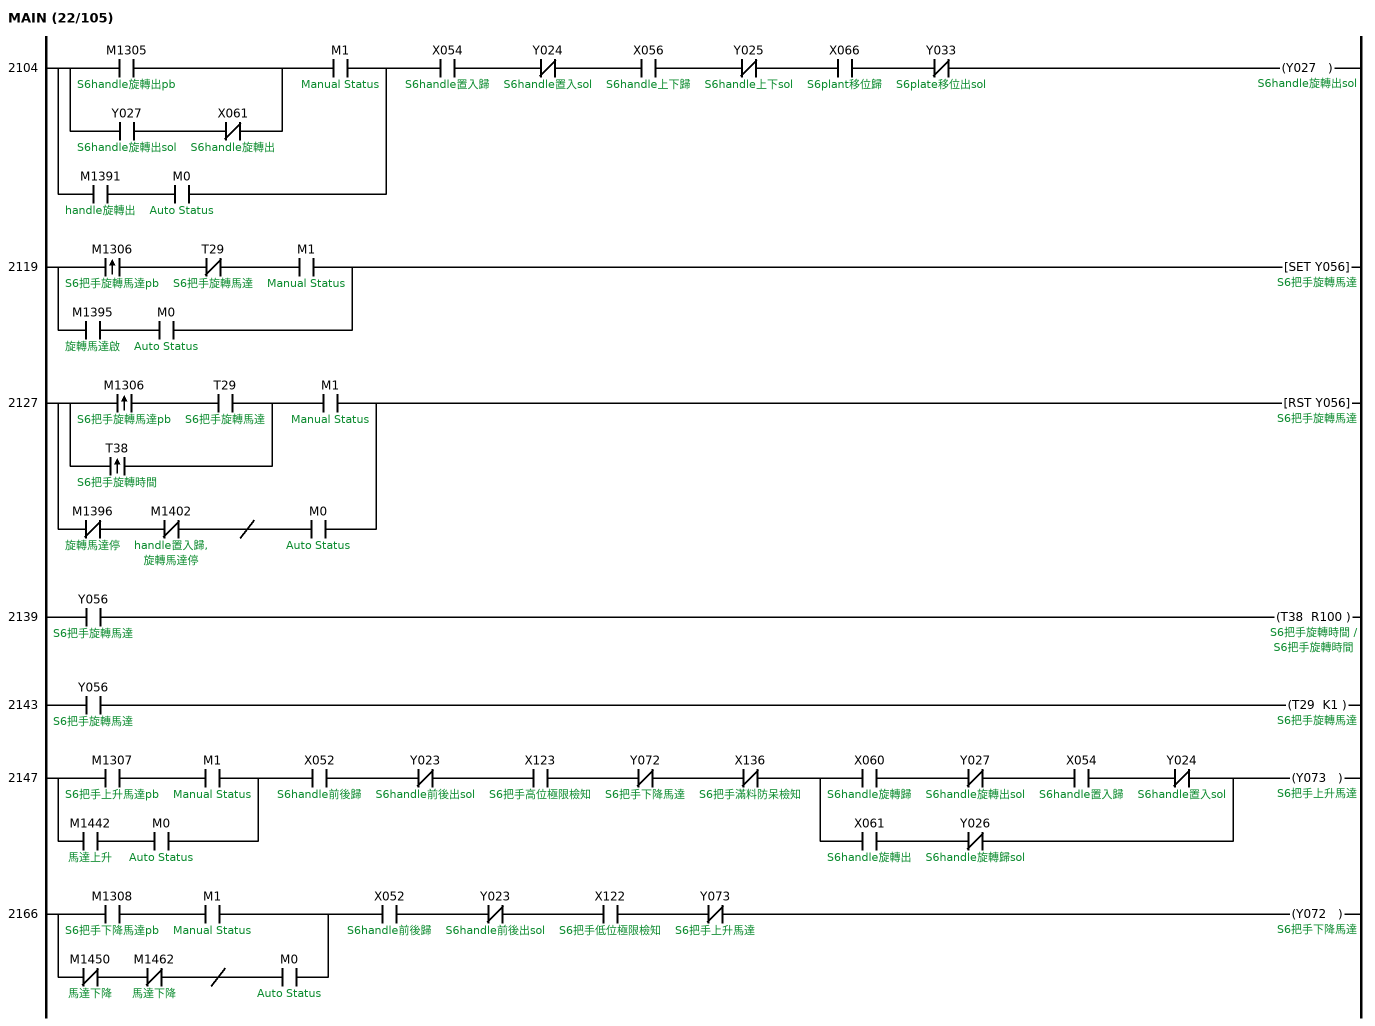
2104  LD      M1305  ; S6handle旋轉出pb
      LD      Y027  ; S6handle旋轉出sol
      ANI     X061  ; S6handle旋轉出
      ORB
      AND     M1  ; Manual Status
      LD      M1391  ; handle旋轉出
      AND     M0  ; Auto Status
      ORB
      AND     X054  ; S6handle置入歸
      ANI     Y024  ; S6handle置入sol
      AND     X056  ; S6handle上下歸
      ANI     Y025  ; S6handle上下sol
      AND     X066  ; S6plant移位歸
      ANI     Y033  ; S6plate移位出sol
      OUT     Y027  ; S6handle旋轉出sol
2119  LDP     M1306  ; S6把手旋轉馬達pb
      ANI     T29  ; S6把手旋轉馬達
      AND     M1  ; Manual Status
      LD      M1395  ; 旋轉馬達啟
      AND     M0  ; Auto Status
      ORB
      SET     Y056  ; S6把手旋轉馬達
2127  LDP     M1306  ; S6把手旋轉馬達pb
      AND     T29  ; S6把手旋轉馬達
      ORP     T38  ; S6把手旋轉時間
      AND     M1  ; Manual Status
      LDI     M1396  ; 旋轉馬達停
      ANI     M1402  ; handle置入歸,旋轉馬達停
      INV
      AND     M0  ; Auto Status
      ORB
      RST     Y056  ; S6把手旋轉馬達
2139  LD      Y056  ; S6把手旋轉馬達
      OUT     T38 R100  ; S6把手旋轉時間 / S6把手旋轉時間
2143  LD      Y056  ; S6把手旋轉馬達
      OUT     T29 K1  ; S6把手旋轉馬達
2147  LD      M1307  ; S6把手上升馬達pb
      AND     M1  ; Manual Status
      LD      M1442  ; 馬達上升
      AND     M0  ; Auto Status
      ORB
      AND     X052  ; S6handle前後歸
      ANI     Y023  ; S6handle前後出sol
      AND     X123  ; S6把手高位極限檢知
      ANI     Y072  ; S6把手下降馬達
      ANI     X136  ; S6把手滿料防呆檢知
      LD      X060  ; S6handle旋轉歸
      ANI     Y027  ; S6handle旋轉出sol
      AND     X054  ; S6handle置入歸
      ANI     Y024  ; S6handle置入sol
      LD      X061  ; S6handle旋轉出
      ANI     Y026  ; S6handle旋轉歸sol
      ORB
      ANB
      OUT     Y073  ; S6把手上升馬達
2166  LD      M1308  ; S6把手下降馬達pb
      AND     M1  ; Manual Status
      LDI     M1450  ; 馬達下降
      ANI     M1462  ; 馬達下降
      INV
      AND     M0  ; Auto Status
      ORB
      AND     X052  ; S6handle前後歸
      ANI     Y023  ; S6handle前後出sol
      AND     X122  ; S6把手低位極限檢知
      ANI     Y073  ; S6把手上升馬達
      OUT     Y072  ; S6把手下降馬達
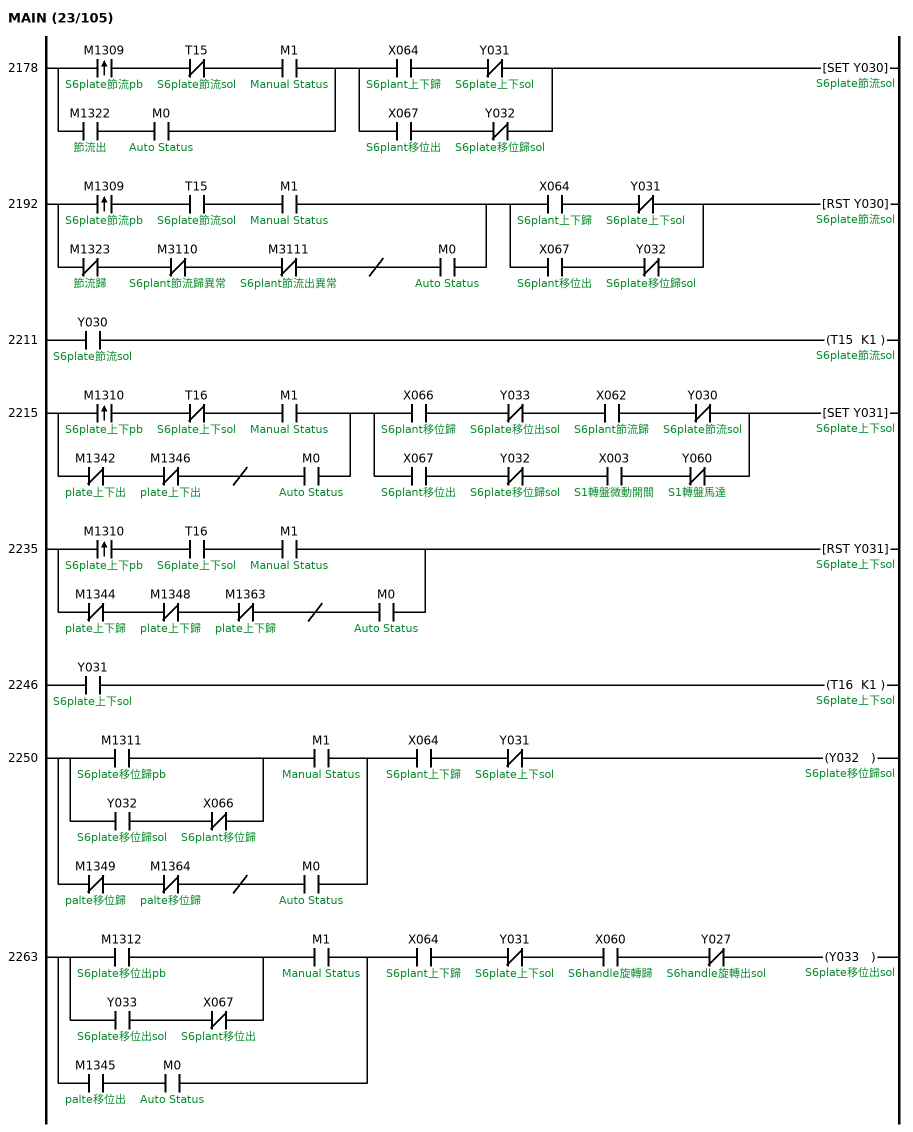
2178  LDP     M1309  ; S6plate節流pb
      ANI     T15  ; S6plate節流sol
      AND     M1  ; Manual Status
      LD      M1322  ; 節流出
      AND     M0  ; Auto Status
      ORB
      LD      X064  ; S6plant上下歸
      ANI     Y031  ; S6plate上下sol
      LD      X067  ; S6plant移位出
      ANI     Y032  ; S6plate移位歸sol
      ORB
      ANB
      SET     Y030  ; S6plate節流sol
2192  LDP     M1309  ; S6plate節流pb
      AND     T15  ; S6plate節流sol
      AND     M1  ; Manual Status
      LDI     M1323  ; 節流歸
      ANI     M3110  ; S6plant節流歸異常
      ANI     M3111  ; S6plant節流出異常
      INV
      AND     M0  ; Auto Status
      ORB
      LD      X064  ; S6plant上下歸
      ANI     Y031  ; S6plate上下sol
      LD      X067  ; S6plant移位出
      ANI     Y032  ; S6plate移位歸sol
      ORB
      ANB
      RST     Y030  ; S6plate節流sol
2211  LD      Y030  ; S6plate節流sol
      OUT     T15 K1  ; S6plate節流sol
2215  LDP     M1310  ; S6plate上下pb
      ANI     T16  ; S6plate上下sol
      AND     M1  ; Manual Status
      LDI     M1342  ; plate上下出
      ANI     M1346  ; plate上下出
      INV
      AND     M0  ; Auto Status
      ORB
      LD      X066  ; S6plant移位歸
      ANI     Y033  ; S6plate移位出sol
      AND     X062  ; S6plant節流歸
      ANI     Y030  ; S6plate節流sol
      LD      X067  ; S6plant移位出
      ANI     Y032  ; S6plate移位歸sol
      AND     X003  ; S1轉盤微動開關
      ANI     Y060  ; S1轉盤馬達
      ORB
      ANB
      SET     Y031  ; S6plate上下sol
2235  LDP     M1310  ; S6plate上下pb
      AND     T16  ; S6plate上下sol
      AND     M1  ; Manual Status
      LDI     M1344  ; plate上下歸
      ANI     M1348  ; plate上下歸
      ANI     M1363  ; plate上下歸
      INV
      AND     M0  ; Auto Status
      ORB
      RST     Y031  ; S6plate上下sol
2246  LD      Y031  ; S6plate上下sol
      OUT     T16 K1  ; S6plate上下sol
2250  LD      M1311  ; S6plate移位歸pb
      LD      Y032  ; S6plate移位歸sol
      ANI     X066  ; S6plant移位歸
      ORB
      AND     M1  ; Manual Status
      LDI     M1349  ; palte移位歸
      ANI     M1364  ; palte移位歸
      INV
      AND     M0  ; Auto Status
      ORB
      AND     X064  ; S6plant上下歸
      ANI     Y031  ; S6plate上下sol
      OUT     Y032  ; S6plate移位歸sol
2263  LD      M1312  ; S6plate移位出pb
      LD      Y033  ; S6plate移位出sol
      ANI     X067  ; S6plant移位出
      ORB
      AND     M1  ; Manual Status
      LD      M1345  ; palte移位出
      AND     M0  ; Auto Status
      ORB
      AND     X064  ; S6plant上下歸
      ANI     Y031  ; S6plate上下sol
      AND     X060  ; S6handle旋轉歸
      ANI     Y027  ; S6handle旋轉出sol
      OUT     Y033  ; S6plate移位出sol
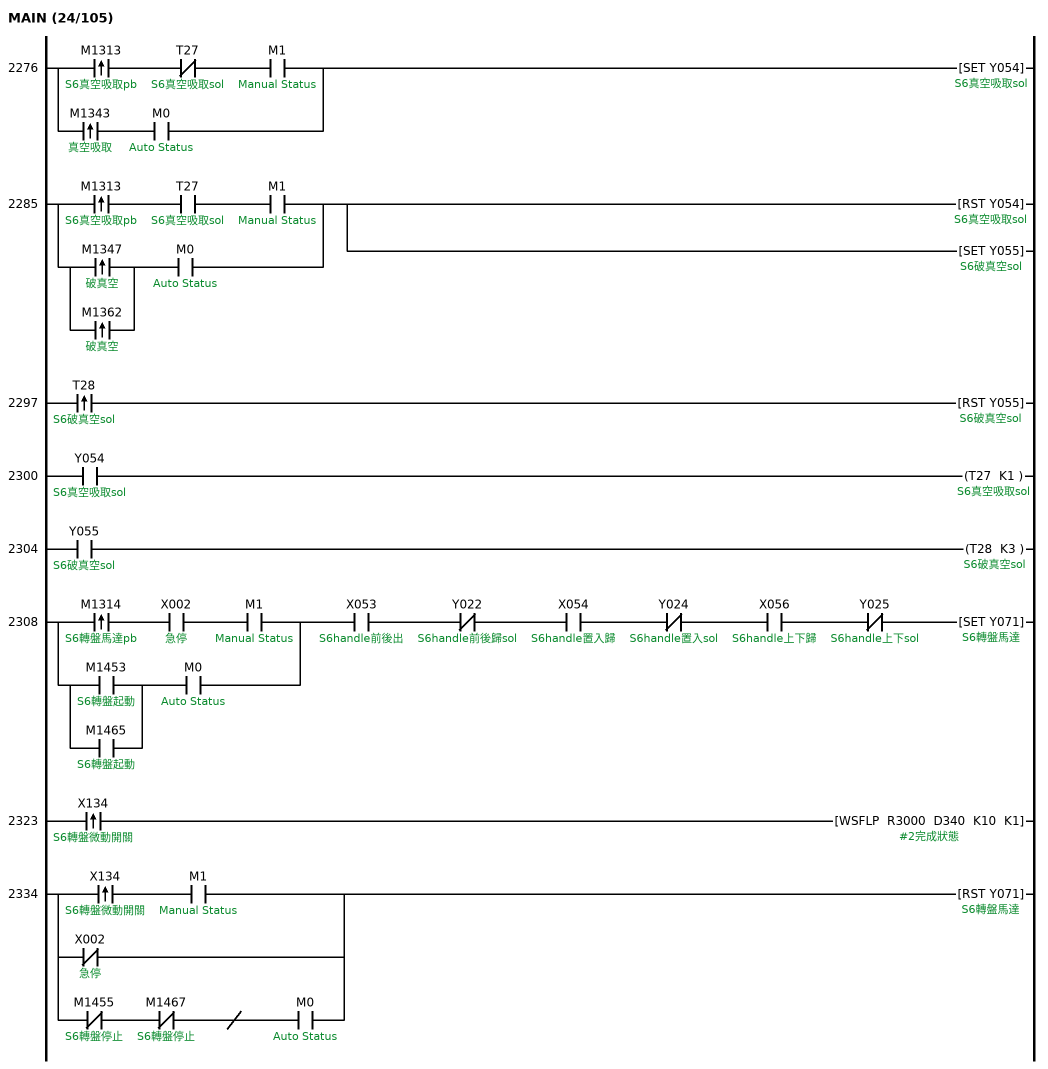
2276  LDP     M1313  ; S6真空吸取pb
      ANI     T27  ; S6真空吸取sol
      AND     M1  ; Manual Status
      LDP     M1343  ; 真空吸取
      AND     M0  ; Auto Status
      ORB
      SET     Y054  ; S6真空吸取sol
2285  LDP     M1313  ; S6真空吸取pb
      AND     T27  ; S6真空吸取sol
      AND     M1  ; Manual Status
      LDP     M1347  ; 破真空
      ORP     M1362  ; 破真空
      AND     M0  ; Auto Status
      ORB
      RST     Y054  ; S6真空吸取sol
      SET     Y055  ; S6破真空sol
2297  LDP     T28  ; S6破真空sol
      RST     Y055  ; S6破真空sol
2300  LD      Y054  ; S6真空吸取sol
      OUT     T27 K1  ; S6真空吸取sol
2304  LD      Y055  ; S6破真空sol
      OUT     T28 K3  ; S6破真空sol
2308  LDP     M1314  ; S6轉盤馬達pb
      AND     X002  ; 急停
      AND     M1  ; Manual Status
      LD      M1453  ; S6轉盤起動
      OR      M1465  ; S6轉盤起動
      AND     M0  ; Auto Status
      ORB
      AND     X053  ; S6handle前後出
      ANI     Y022  ; S6handle前後歸sol
      AND     X054  ; S6handle置入歸
      ANI     Y024  ; S6handle置入sol
      AND     X056  ; S6handle上下歸
      ANI     Y025  ; S6handle上下sol
      SET     Y071  ; S6轉盤馬達
2323  LDP     X134  ; S6轉盤微動開關
      WSFLP   R3000 D340 K10 K1
2334  LDP     X134  ; S6轉盤微動開關
      AND     M1  ; Manual Status
      ORI     X002  ; 急停
      LDI     M1455  ; S6轉盤停止
      ANI     M1467  ; S6轉盤停止
      INV
      AND     M0  ; Auto Status
      ORB
      RST     Y071  ; S6轉盤馬達
